			// at this point we are not currently "parsing" a known type from the string, therfore the next character should 
			// decide what type is next. 
		
			IF Path[currentCharacterPositionInPath] = DOLLAR_SIGN THEN
				
				// i.e. the following string $.myValue would indicate that we are here.
				//                           ^                                         
				// as such, we do not need to take any action.  We already create a root element at the start, so this is an 
				// optional character which they do not need to supply. 				
				
			ELSIF Path[currentCharacterPositionInPath] = PERIOD THEN
				
				// i.e. the following string $.myValue would indicate that we are here.
				//                            ^                                        
				// as such, we do not need to take any action.  
				
			ELSIF Path[currentCharacterPositionInPath] = LEFT_SQUARE_BRACKET THEN
				
				// i.e. the following string $.myValue[1].['myProperty'] would indicate that we could be at the start of one of two types
				//                                    ^   ^                                      
				// as such, we mark that we could be either a property or array and continue				
				currentlyParsingType := BRACKET_NOTATION_PROPERTY_OR_ARRAY;				
				
			ELSIF Path[currentCharacterPositionInPath] = RIGHT_SQUARE_BRACKET THEN
				
				// This would indicate a failed parse as this should not happen.
				JsonPathVisitor.InvalidSyntaxFound(RIGHT_SQUARE_BRACKET, currentCharacterPositionInPath);
				
			ELSIF Path[currentCharacterPositionInPath] = SINGLE_QUOTE THEN
				
				// This would indicate a failed parse as this should not happen.
				JsonPathVisitor.InvalidSyntaxFound(SINGLE_QUOTE, currentCharacterPositionInPath);
				
			ELSE
				
				// i.e. the following string $.myValue[1].['myProperty'] would indicate that we could be at the start of a property
				//                             ^                      
				currentlyParsingType := DOT_NOTATION_PROPERTY;
				currentElementStart := currentCharacterPositionInPath;	
		
			END_IF
			
		DOT_NOTATION_PROPERTY:
		
			IF Path[currentCharacterPositionInPath] = PERIOD OR Path[currentCharacterPositionInPath] = LEFT_SQUARE_BRACKET OR Path[currentCharacterPositionInPath] = NULL THEN
				
				currentElementEnd := currentCharacterPositionInPath - 1;
				
				currentElementLength := 1 + currentElementEnd - currentElementStart;
				memset(ADR(elementText),0,SIZEOF(elementText));
				memcpy(ADR(elementText),ADR(Path[currentElementStart]),currentElementLength);
		
				JsonPathVisitor.PropertyFound(elementText);
				
				currentlyParsingType := NOTHING;
				CONTINUE;
				
			END_IF
			
		BRACKET_NOTATION_PROPERTY_OR_ARRAY:
		
			IF Path[currentCharacterPositionInPath] = SINGLE_QUOTE THEN
				currentlyParsingType := BRACKET_NOTATION_PROPERTY_ELEMENT;
				currentElementStart := currentCharacterPositionInPath + 1;			
			ELSE
				currentlyParsingType := BRACKET_NOTATION_ARRAY_ELEMENT;
				currentElementStart := currentCharacterPositionInPath;			
			END_IF
			
		BRACKET_NOTATION_PROPERTY_ELEMENT:
		
			IF Path[currentCharacterPositionInPath] = SINGLE_QUOTE THEN
				
				currentElementEnd := currentCharacterPositionInPath - 1;

				currentElementLength := 1 + currentElementEnd - currentElementStart;
				memset(ADR(elementText),0,SIZEOF(elementText));
				memcpy(ADR(elementText),ADR(Path[currentElementStart]),currentElementLength);
				
				JsonPathVisitor.PropertyFound(elementText);
			
				currentlyParsingType := NOTHING;
						
			END_IF
			
		BRACKET_NOTATION_ARRAY_ELEMENT:
		
			IF Path[currentCharacterPositionInPath] = RIGHT_SQUARE_BRACKET THEN
				
				currentElementEnd := currentCharacterPositionInPath - 1;
				
				currentElementLength := 1 + currentElementEnd - currentElementStart;
				memset(ADR(elementText),0,SIZEOF(elementText));
				memcpy(ADR(elementText),ADR(Path[currentElementStart]),currentElementLength);
				
				JsonPathVisitor.ArrayIndexFound(STRING_TO_UDINT(elementText));		
				currentlyParsingType := NOTHING;
						
			END_IF
			

	END_CASE
	
	currentCharacterPositionInPath := currentCharacterPositionInPath + 1;
	
UNTIL endOfRepeat 
END_REPEAT

JsonPathVisitor.EndOfParse();
END_METHOD

END_FUNCTION_BLOCK

// mobject-json/_Internal/JsonPathVisitor/I_JsonPathVisitor
INTERFACE I_JsonPathVisitor EXTENDS __System.IQueryInterface

METHOD ArrayIndexFound
VAR_INPUT
	Index : UDINT;
END_VAR
END_METHOD

METHOD EndOfParse
VAR_INPUT
END_VAR
END_METHOD

METHOD InvalidSyntaxFound
VAR_INPUT
	Character : BYTE;
	Position : UDINT;
END_VAR
END_METHOD

METHOD PropertyFound
VAR_INPUT
	Name : T_MAXSTRING;
END_VAR
END_METHOD

METHOD StartOfParse
VAR_INPUT
END_VAR
END_METHOD

END_INTERFACE

// mobject-json/_Internal/JsonPathVisitor/JsonDomNavigator
{attribute 'linkalways'} 
{attribute 'no_explicit_call' := 'This FB is a CLASS and must be accessed using methods or properties'}
{attribute 'enable_dynamic_creation'}
FUNCTION_BLOCK JsonDomNavigator IMPLEMENTS I_JsonPathVisitor
VAR
	jsonDomParser : REFERENCE TO JsonDomParser;
	currentJsonPosition : SJsonValue;
	_currentNode : SJsonValue;
END_VAR

METHOD FB_init : BOOL
VAR_INPUT
	bInitRetains : BOOL; // if TRUE, the retain variables are initialized (warm start / cold start)
	bInCopyCode : BOOL;  // if TRUE, the instance afterwards gets moved into the copy code (online change)
	JsonDomParser : REFERENCE TO JsonDomParser;
END_VAR
THIS^.jsonDomParser REF= JsonDomParser;
END_METHOD

METHOD ArrayIndexFound
VAR_INPUT
	Index : UDINT;
END_VAR
currentJsonPosition := jsonDomParser.GetArrayValueByIdx(currentJsonPosition, Index);
END_METHOD

PROPERTY PUBLIC CurrentNode : SJsonValue
GET
CurrentNode := _currentNode;
END_GET
END_PROPERTY

METHOD EndOfParse
VAR_INPUT
END_VAR
_currentNode := currentJsonPosition;
END_METHOD

METHOD InvalidSyntaxFound
VAR_INPUT
	Character : BYTE;
	Position : UDINT;
END_VAR
currentJsonPosition := 0;
END_METHOD

METHOD PropertyFound
VAR_INPUT
	Name : T_MAXSTRING;
END_VAR
currentJsonPosition := jsonDomParser.FindMember(currentJsonPosition,Name);
END_METHOD

METHOD StartOfParse
VAR_INPUT
END_VAR
currentJsonPosition := jsonDomParser.GetDocumentRoot();
END_METHOD

END_FUNCTION_BLOCK

// mobject-json/_Internal/JsonPathVisitor/JsonDomCreator
{attribute 'linkalways'} 
{attribute 'no_explicit_call' := 'This FB is a CLASS and must be accessed using methods or properties'}
{attribute 'enable_dynamic_creation'}
FUNCTION_BLOCK JsonDomCreator IMPLEMENTS I_JsonPathVisitor
VAR
	jsonDomParser : REFERENCE TO JsonDomParser;
	currentJsonPosition : SJsonValue;
	_currentNode : SJsonValue;
END_VAR

METHOD FB_init : BOOL
VAR_INPUT
	bInitRetains : BOOL; // if TRUE, the retain variables are initialized (warm start / cold start)
	bInCopyCode : BOOL;  // if TRUE, the instance afterwards gets moved into the copy code (online change)
	JsonDomParser : REFERENCE TO JsonDomParser;
END_VAR
THIS^.jsonDomParser REF= JsonDomParser;
END_METHOD

METHOD PRIVATE PadStartOfArray : SJsonValue
VAR_INPUT
	Index : UDINT;
	ArrayPosition : SJsonValue;
END_VAR
VAR
	i : UDINT;
	arrayValueLocation : SJsonValue;
END_VAR
FOR i := 0 TO Index DO
		
	arrayValueLocation := jsonDomParser.GetArrayValueByIdx(ArrayPosition, Index);
	IF arrayValueLocation <> 0 THEN
		CONTINUE;
	END_IF
	
	arrayValueLocation := jsonDomParser.PushbackNullValue(ArrayPosition);

END_FOR

PadStartOfArray := arrayValueLocation;
END_METHOD

METHOD ArrayIndexFound
VAR_INPUT
	Index : UDINT;
END_VAR
VAR
	memberLocation : SJsonValue;
	i : UDINT;
END_VAR
IF jsonDomParser.IsArray(currentJsonPosition) THEN
	
	memberLocation := jsonDomParser.GetArrayValueByIdx(currentJsonPosition, Index);
	
	IF memberLocation <> 0 THEN
		currentJsonPosition := memberLocation;
		RETURN;
	END_IF
	
	currentJsonPosition := PadStartOfArray(Index, currentJsonPosition);

else
	
	memberLocation := jsonDomParser.SetArray(currentJsonPosition,0);
	currentJsonPosition := PadStartOfArray(Index, memberLocation);
	
END_IF
END_METHOD

PROPERTY PUBLIC CurrentNode : SJsonValue
GET
CurrentNode := _currentNode;
END_GET
END_PROPERTY

METHOD EndOfParse
VAR_INPUT
END_VAR
_currentNode := currentJsonPosition;
END_METHOD

METHOD InvalidSyntaxFound
VAR_INPUT
	Character : BYTE;
	Position : UDINT;
END_VAR
currentJsonPosition := 0;
END_METHOD

METHOD PropertyFound
VAR_INPUT
	Name : T_MAXSTRING;
END_VAR
VAR
	memberLocation : SJsonValue;
END_VAR
memberLocation := jsonDomParser.FindMember(currentJsonPosition,Name);

IF memberLocation <> 0 THEN
	currentJsonPosition := memberLocation;
	RETURN;
END_IF

currentJsonPosition := jsonDomParser.AddNullMember(currentJsonPosition,Name);
END_METHOD

METHOD StartOfParse
VAR_INPUT
END_VAR
currentJsonPosition := jsonDomParser.GetDocumentRoot();
END_METHOD

END_FUNCTION_BLOCK

// mobject-json/_Internal/JsonDeserializerNode/JsonDeserializerNode
{attribute 'linkalways'} 
{attribute 'no_explicit_call' := 'This FB is a CLASS and must be accessed using methods or properties'}
{attribute 'enable_dynamic_creation'}
FUNCTION_BLOCK JsonDeserializerNode EXTENDS Disposable IMPLEMENTS I_Deserializer
VAR	
	parent : I_JsonDeserializer;
	jsonParser : REFERENCE TO JsonDomParser;
	root : SJsonValue;
	garbageCollector : I_DeserializerGarbageCollector;
	nullNode : I_Deserializer;
	errorFactory : DeserializationErrorFactory;
END_VAR

METHOD FB_init : BOOL
VAR_INPUT
	bInitRetains : BOOL; // if TRUE, the retain variables are initialized (warm start / cold start)
	bInCopyCode : BOOL;  // if TRUE, the instance afterwards gets moved into the copy code (online change)
	ParentJsonDeserializer : I_JsonDeserializer;
	ParentJsonDomParser : REFERENCE TO JsonDomParser;
	NodeRoot : SJsonValue;
	ParentGarbageCollector : I_DeserializerGarbageCollector;
	ParentNullDeserializer : I_Deserializer;
END_VAR
THIS^.parent := ParentJsonDeserializer;
THIS^.jsonParser REF= ParentJsonDomParser;
THIS^.root := NodeRoot;
THIS^.garbageCollector := ParentGarbageCollector;
THIS^.nullNode := ParentNullDeserializer;

ParentGarbageCollector.Register(THIS^);
END_METHOD

METHOD PROTECTED CreateArrayForwardEnumerator : I_DeserializerArrayForwardEnumerator
VAR_INPUT
	DeserializerRoot : SJsonValue;
END_VAR
VAR 
	pForwardEnumerator : POINTER TO JsonDeserializerArrayForwardEnumerator;
END_VAR
pForwardEnumerator := __NEW(JsonDeserializerArrayForwardEnumerator(
	ParentJsonDeserializer := parent,
	ParentJsonDomParser := jsonParser, 
	NodeRoot := DeserializerRoot, 
	ParentGarbageCollector := garbageCollector, 
	ParentNullDeserializer := nullNode
));

CreateArrayForwardEnumerator := pForwardEnumerator^;
END_METHOD

METHOD PROTECTED CreateDeserializer : I_Deserializer
VAR_INPUT
	DeserializerRoot : SJsonValue;
END_VAR
VAR 
	pNode : POINTER TO JsonDeserializerNode;
END_VAR
pNode := __NEW(JsonDeserializerNode(
	ParentJsonDeserializer := parent,
	ParentJsonDomParser := jsonParser, 
	NodeRoot := DeserializerRoot, 
	ParentGarbageCollector := garbageCollector, 
	ParentNullDeserializer := nullNode
));

CreateDeserializer := pNode^;
END_METHOD

METHOD PROTECTED CreateObjectForwardEnumerator : I_DeserializerObjectForwardEnumerator
VAR_INPUT
	DeserializerRoot : SJsonValue;
END_VAR
VAR 
	pForwardEnumerator : POINTER TO JsonDeserializerObjectForwardEnumerator;
END_VAR
pForwardEnumerator := __NEW(JsonDeserializerObjectForwardEnumerator(
	ParentJsonDeserializer := parent,
	ParentJsonDomParser := jsonParser, 
	NodeRoot := DeserializerRoot, 
	ParentGarbageCollector := garbageCollector, 
	ParentNullDeserializer := nullNode
));

CreateObjectForwardEnumerator := pForwardEnumerator^;
END_METHOD

METHOD PROTECTED TryGetMember : BOOL
VAR_INPUT
	MemberName : T_MAXSTRING;
	Member : REFERENCE TO SJsonValue;
	Feedback : I_DeserializerFeedback;
END_VAR
VAR
	localMember : SJsonValue;
	error : I_Error;
END_VAR
IF MemberName = '' THEN
	error := errorFactory.CreateInvalidKeyError();
	Feedback.LogError(error);
	RETURN;
END_IF

localMember := jsonParser.FindMember(root, MemberName);

IF localMember = 0 THEN
	error := errorFactory.CreateMissingKeyError(MemberName);
	Feedback.LogError(error);
	RETURN;
END_IF

Member := localMember;
TryGetMember := TRUE;
END_METHOD

METHOD PROTECTED TryReadBool : BOOL
VAR_INPUT
	JsonValue : SJsonValue;
	Destination : ANY;
END_VAR
VAR
	_BOOL : BOOL;
END_VAR
IF jsonValue = 0 THEN
	RETURN;
END_IF

IF jsonParser.IsBool(jsonValue) THEN
	_BOOL := jsonParser.GetBool(jsonValue);
	TryReadBool := TryConvert_BOOL_TO_DESTINATION(_BOOL,Destination);
	RETURN;
END_IF
END_METHOD

METHOD PROTECTED TryReadNumber : BOOL
VAR_INPUT
	JsonValue : SJsonValue;
	Destination : ANY;
END_VAR
VAR
	_DINT : DINT;
	_LINT : LINT;
	_UDINT : UDINT;
	_ULINT : ULINT;
	_LREAL : LREAL;
END_VAR
IF jsonValue = 0 THEN
	RETURN;
END_IF

IF jsonParser.IsInt(jsonValue) THEN
	_DINT := jsonParser.GetInt(jsonValue);
	TryReadNumber := TryConvert_DINT_TO_DESTINATION(_DINT,Destination);
	RETURN;
END_IF

IF jsonParser.IsInt64(jsonValue) THEN
	_LINT := jsonParser.GetInt64(jsonValue);
	TryReadNumber := TryConvert_LINT_TO_DESTINATION(_LINT,Destination);
	RETURN;
END_IF

IF jsonParser.IsUInt(jsonValue) THEN
	_UDINT := jsonParser.GetUInt(jsonValue);
	TryReadNumber := TryConvert_UDINT_TO_DESTINATION(_UDINT,Destination);
	RETURN;
END_IF

IF jsonParser.IsUInt64(jsonValue) THEN
	_ULINT := jsonParser.GetUInt64(jsonValue);
	TryReadNumber := TryConvert_ULINT_TO_DESTINATION(_ULINT,Destination);
	RETURN;
END_IF

IF jsonParser.IsDouble(jsonValue) THEN
	_LREAL := jsonParser.GetDouble(jsonValue);
	TryReadNumber := TryConvert_LREAL_TO_DESTINATION(_LREAL,Destination);
	RETURN;
END_IF
END_METHOD

METHOD PROTECTED TryReadString : BOOL
VAR_INPUT
	JsonValue : SJsonValue;
	Destination : REFERENCE TO STRING;
END_VAR
IF jsonValue = 0 THEN
	RETURN;
END_IF

IF jsonParser.IsString(jsonValue) THEN
	IF (jsonParser.CopyString(jsonValue,Destination,DINT_TO_UDINT(SIZEOF(Destination))) > 0) THEN;
		TryReadString := TRUE;
		RETURN;
	END_IF
END_IF
END_METHOD

METHOD PUBLIC Clone : I_Deserializer
VAR
	pClone : POINTER TO JsonDeserializer;
	jsonSize : UDINT;
	pJsonString : POINTER TO STRING;
END_VAR
pClone := __NEW(JsonDeserializer);
Clone := pClone^;

jsonSize := jsonParser.GetJsonLength(root);

IF jsonSize = 0 THEN
	// no further cloning to do. 
	RETURN;
END_IF

pJsonString := __NEW(BYTE, jsonSize);

IF jsonParser.CopyJson(root, pJsonString^, jsonSize) = 0 THEN
	__DELETE(pJsonString);
	RETURN;
END_IF

pClone^.TryLoad(pJsonString^);
__DELETE(pJsonString);
END_METHOD

METHOD Dispose
VAR
END_VAR
garbageCollector.Deregister(THIS^);
super^.Dispose();
END_METHOD

METHOD GetArray : I_Deserializer
IF NOT jsonParser.IsArray(root) THEN
	GetArray := nullNode;
	RETURN;
END_IF

GetArray := CreateDeserializer(root);
END_METHOD

METHOD GetArrayEnumerator : I_DeserializerArrayForwardEnumerator
VAR_INPUT
END_VAR
GetArrayEnumerator := CreateArrayForwardEnumerator(root);
END_METHOD

METHOD GetElementByIndex : I_Deserializer
VAR_INPUT
	Index : UDINT;
END_VAR
VAR
	newRoot : SJsonValue;
END_VAR
IF NOT jsonParser.IsArray(root) THEN
	GetElementByIndex := nullNode;
	RETURN;
END_IF

newRoot := jsonParser.GetArrayValueByIdx(root, Index);

IF newRoot = 0 THEN
	GetElementByIndex := nullNode;
	RETURN;
END_IF

GetElementByIndex := CreateDeserializer(newRoot);
END_METHOD

METHOD GetKeyArray : I_Deserializer
VAR_INPUT
	Key : T_MAXSTRING;
END_VAR
VAR
	member : SJsonValue;
END_VAR
IF key = '' THEN
	RETURN;
END_IF

member := jsonParser.FindMember(root,Key);

IF member = 0 THEN
	GetKeyArray := nullNode;
	RETURN;
END_IF

IF NOT jsonParser.IsArray(member) THEN
	GetKeyArray := nullNode;
	RETURN;
END_IF

GetKeyArray := CreateDeserializer(member);
END_METHOD

METHOD GetKeyObject : I_Deserializer
VAR_INPUT
	Key : T_MAXSTRING;
END_VAR
VAR
	newRoot : SJsonValue;
END_VAR
newRoot := jsonParser.FindMember(root, Key);

IF newRoot = 0 THEN
	GetKeyObject := nullNode;
	RETURN;
END_IF

GetKeyObject := CreateDeserializer(newRoot);
END_METHOD

METHOD GetObject : I_Deserializer
IF NOT jsonParser.IsObject(root) THEN
	GetObject := nullNode;
	RETURN;
END_IF

GetObject := CreateDeserializer(root);
END_METHOD

METHOD GetObjectEnumerator : I_DeserializerObjectForwardEnumerator
VAR_INPUT
END_VAR
GetObjectEnumerator := CreateObjectForwardEnumerator(root);
END_METHOD

METHOD GetValue : I_Deserializer
VAR
	newRoot : SJsonValue;
END_VAR
newRoot := jsonParser.GetMemberValue(root);

IF newRoot = 0 THEN
	GetValue := nullNode;
	RETURN;
END_IF

GetValue := CreateDeserializer(newRoot);
END_METHOD

METHOD TryDeserializeKeyToObject : BOOL
VAR_INPUT
	Key : T_MAXSTRING;
	Object : I_Deserializable;
	Feedback : I_DeserializerFeedback;
END_VAR
VAR
	member : SJsonValue;
	error : I_Error;
	deserializer : I_Deserializer;
END_VAR
IF NOT TryGetMember(Key, member, Feedback) THEN
	RETURN;
END_IF

deserializer := CreateDeserializer(member);
TryDeserializeKeyToObject := Object.TryDeserializeFrom(deserializer, Feedback);
END_METHOD

METHOD TryDeserializeToObject : BOOL
VAR_INPUT
	Object : I_Deserializable;
	Feedback : I_DeserializerFeedback;
END_VAR
TryDeserializeToObject := Object.TryDeserializeFrom(THIS^, Feedback);
END_METHOD

METHOD TryGetBase64 : BOOL
VAR_INPUT
	pBytes : POINTER TO BYTE;
	nBytes : DINT;
	Feedback : I_DeserializerFeedback;
END_VAR
VAR
	error : I_Error;
END_VAR
IF NOT jsonParser.IsBase64(root) THEN
	error := errorFactory.CreateIncorrectTypeError('Base64');
	Feedback.LogError(error);
	RETURN;
END_IF

jsonParser.GetBase64(root, pBytes, nBytes);
TryGetBase64 := TRUE;
END_METHOD

METHOD TryGetBool : BOOL
VAR_INPUT
	Destination : REFERENCE TO BOOL;
	Feedback : I_DeserializerFeedback;
END_VAR
VAR
	value : BOOL;
	error : I_Error;
END_VAR
IF NOT TryReadBool(root, value) THEN
	error := errorFactory.CreateIncorrectTypeError('BOOL');
	Feedback.LogError(error);
	RETURN;
END_IF

Destination := value;
TryGetBool := TRUE;
END_METHOD

METHOD TryGetByte : BOOL
VAR_INPUT
	Destination : REFERENCE TO BYTE;
	Feedback : I_DeserializerFeedback;
END_VAR
VAR
	value : BYTE;
	error : I_Error;
END_VAR
IF NOT TryReadNumber(root, value) THEN
	error := errorFactory.CreateIncorrectTypeError('BYTE');
	Feedback.LogError(error);
	RETURN;
END_IF

Destination := value;
TryGetByte := TRUE;
END_METHOD

METHOD TryGetDateTime : BOOL
VAR_INPUT
	Destination : REFERENCE TO DATE_AND_TIME;
	Feedback : I_DeserializerFeedback;
END_VAR
VAR
	error : I_Error;
END_VAR
IF NOT jsonParser.IsISO8601TimeFormat(root) THEN
	error := errorFactory.CreateIncorrectTypeError('DATE_AND_TIME');
	Feedback.LogError(error);
	RETURN;
END_IF

Destination := jsonParser.GetDateTime(root);
TryGetDateTime := TRUE;
END_METHOD

METHOD TryGetDcTime : BOOL
VAR_INPUT
	Destination : REFERENCE TO DCTIME;
	Feedback : I_DeserializerFeedback;
END_VAR
VAR
	error : I_Error;
END_VAR
IF NOT jsonParser.IsISO8601TimeFormat(root) THEN
	error := errorFactory.CreateIncorrectTypeError('DCTIME');
	Feedback.LogError(error);
	RETURN;
END_IF

Destination := jsonParser.GetDcTime(root);
TryGetDcTime := TRUE;
END_METHOD

METHOD TryGetDint : BOOL
VAR_INPUT
	Destination : REFERENCE TO DINT;
	Feedback : I_DeserializerFeedback;
END_VAR
VAR
	value : DINT;
	error : I_Error;
END_VAR
IF NOT TryReadNumber(root, value) THEN
	error := errorFactory.CreateIncorrectTypeError('DINT');
	Feedback.LogError(error);
	RETURN;
END_IF

Destination := value;
TryGetDint := TRUE;
END_METHOD

METHOD TryGetDword : BOOL
VAR_INPUT
	Destination : REFERENCE TO DWORD;
	Feedback : I_DeserializerFeedback;
END_VAR
VAR
	value : DWORD;
	error : I_Error;
END_VAR
IF NOT TryReadNumber(root, value) THEN
	error := errorFactory.CreateIncorrectTypeError('DWORD');
	Feedback.LogError(error);
	RETURN;
END_IF

Destination := value;
TryGetDword := TRUE;
END_METHOD

METHOD TryGetFileTime : BOOL
VAR_INPUT
	Destination : REFERENCE TO FILETIME;
	Feedback : I_DeserializerFeedback;
END_VAR
VAR
	error : I_Error;
END_VAR
IF NOT jsonParser.IsISO8601TimeFormat(root) THEN
	error := errorFactory.CreateIncorrectTypeError('FILETIME');
	Feedback.LogError(error);
	RETURN;
END_IF

Destination := jsonParser.GetFileTime(root);
TryGetFileTime := TRUE;
END_METHOD

METHOD TryGetHexAsBytes : BOOL
VAR_INPUT
	pBytes : POINTER TO BYTE;
	nBytes : DINT;
	Feedback : I_DeserializerFeedback;
END_VAR
VAR
	error : I_Error;
END_VAR
IF NOT jsonParser.IsHexBinary(root) THEN
	error := errorFactory.CreateIncorrectTypeError('HexBinary');
	Feedback.LogError(error);
	RETURN;
END_IF

jsonParser.GetHexBinary(root, pBytes, nBytes);
TryGetHexAsBytes := TRUE;
END_METHOD

METHOD TryGetInt : BOOL
VAR_INPUT
	Destination : REFERENCE TO INT;
	Feedback : I_DeserializerFeedback;
END_VAR
VAR
	value : INT;
	error : I_Error;
END_VAR
IF NOT TryReadNumber(root, value) THEN
	error := errorFactory.CreateIncorrectTypeError('INT');
	Feedback.LogError(error);
	RETURN;
END_IF

Destination := value;
TryGetInt := TRUE;
END_METHOD

METHOD TryGetKeyBase64 : BOOL
VAR_INPUT
	Key : T_MAXSTRING;
	pBytes : POINTER TO BYTE;
	nBytes : DINT;
	Feedback : I_DeserializerFeedback;
END_VAR
VAR
	member : SJsonValue;
	error : I_Error;
END_VAR
IF NOT TryGetMember(Key, member, Feedback) THEN
	RETURN;
END_IF

IF NOT jsonParser.IsBase64(member) THEN
	error := errorFactory.CreateIncorrectKeyTypeError('Base64',Key);
	Feedback.LogError(error);
	RETURN;
END_IF

jsonParser.GetBase64(member, pBytes, nBytes);
TryGetKeyBase64 := TRUE;
END_METHOD

METHOD TryGetKeyBool : BOOL
VAR_INPUT
	Key : T_MAXSTRING;
	Destination : REFERENCE TO BOOL;
	Feedback : I_DeserializerFeedback;
END_VAR
VAR
	member : SJsonValue;
	value : BOOL;
	error : I_Error;
END_VAR
IF NOT TryGetMember(Key, member, Feedback) THEN
	RETURN;
END_IF

IF NOT TryReadBool(member, value) THEN
	error := errorFactory.CreateIncorrectKeyTypeError('BOOL',Key);
	Feedback.LogError(error);
	RETURN;
END_IF

Destination := value;
TryGetKeyBool := TRUE;
END_METHOD

METHOD TryGetKeyByte : BOOL
VAR_INPUT
	Key : T_MAXSTRING;
	Destination : REFERENCE TO BYTE;
	Feedback : I_DeserializerFeedback;
END_VAR
VAR
	value : BYTE;
	member : SJsonValue;
	error : I_Error;
END_VAR
IF NOT TryGetMember(Key, member, Feedback) THEN
	RETURN;
END_IF

IF NOT TryReadNumber(member, value) THEN
	error := errorFactory.CreateIncorrectKeyTypeError('BYTE',Key);
	Feedback.LogError(error);
	RETURN;
END_IF

Destination := value;
TryGetKeyByte := TRUE;
END_METHOD

METHOD TryGetKeyDateTime : BOOL
VAR_INPUT
	Key : T_MAXSTRING;
	Destination : REFERENCE TO DATE_AND_TIME;
	Feedback : I_DeserializerFeedback;
END_VAR
VAR
	member : SJSonValue;
	error : I_Error;
END_VAR
IF NOT TryGetMember(Key, member, Feedback) THEN
	RETURN;
END_IF

IF NOT jsonParser.IsISO8601TimeFormat(member) THEN
	error := errorFactory.CreateIncorrectKeyTypeError('DATE_AND_TIME',Key);
	Feedback.LogError(error);
	RETURN;
END_IF

Destination := jsonParser.GetDateTime(member);
TryGetKeyDateTime := TRUE;
END_METHOD

METHOD TryGetKeyDcTime : BOOL
VAR_INPUT
	Key : T_MAXSTRING;
	Destination : REFERENCE TO DCTIME;
	Feedback : I_DeserializerFeedback;
END_VAR
VAR
	member : SJSonValue;
	error : I_Error;
END_VAR
IF NOT TryGetMember(Key, member, Feedback) THEN
	RETURN;
END_IF

IF NOT jsonParser.IsISO8601TimeFormat(member) THEN
	error := errorFactory.CreateIncorrectKeyTypeError('DCTIME',Key);
	Feedback.LogError(error);
	RETURN;
END_IF

Destination := jsonParser.GetDcTime(member);
TryGetKeyDcTime := TRUE;
END_METHOD

METHOD TryGetKeyDint : BOOL
VAR_INPUT
	Key : T_MAXSTRING;
	Destination : REFERENCE TO DINT;
	Feedback : I_DeserializerFeedback;
END_VAR
VAR
	member : SJsonValue;
	value : DINT;
	error : I_Error;
END_VAR
IF NOT TryGetMember(Key, member, Feedback) THEN
	RETURN;
END_IF

IF NOT TryReadNumber(member, value) THEN
	error := errorFactory.CreateIncorrectKeyTypeError('DINT',Key);
	Feedback.LogError(error);
	RETURN;
END_IF

Destination := value;
TryGetKeyDint := TRUE;
END_METHOD

METHOD TryGetKeyDword : BOOL
VAR_INPUT
	Key : T_MAXSTRING;
	Destination : REFERENCE TO DWORD;
	Feedback : I_DeserializerFeedback;
END_VAR
VAR
	member : SJsonValue;
	value : DWORD;
	error : I_Error;
END_VAR
IF NOT TryGetMember(Key, member, Feedback) THEN
	RETURN;
END_IF

IF NOT TryReadNumber(member, value) THEN
	error := errorFactory.CreateIncorrectKeyTypeError('DWORD',Key);
	Feedback.LogError(error);
	RETURN;
END_IF

Destination := value;
TryGetKeyDword := TRUE;
END_METHOD

METHOD TryGetKeyFileTime : BOOL
VAR_INPUT
	Key : T_MAXSTRING;
	Destination : REFERENCE TO FILETIME;
	Feedback : I_DeserializerFeedback;
END_VAR
VAR
	member : SJSonValue;
	error : I_Error;
END_VAR
IF NOT TryGetMember(Key, member, Feedback) THEN
	RETURN;
END_IF

IF NOT jsonParser.IsISO8601TimeFormat(member) THEN
	error := errorFactory.CreateIncorrectKeyTypeError('FILETIME',Key);
	Feedback.LogError(error);
	RETURN;
END_IF

Destination := jsonParser.GetFileTime(member);
TryGetKeyFileTime := TRUE;
END_METHOD

METHOD TryGetKeyHexAsBytes : BOOL
VAR_INPUT
	Key : T_MAXSTRING;
	pBytes : POINTER TO BYTE;
	nBytes : DINT;
	Feedback : I_DeserializerFeedback;
END_VAR
VAR
	member : SJsonValue;
	error : I_Error;
END_VAR
IF NOT TryGetMember(Key, member, Feedback) THEN
	RETURN;
END_IF

IF NOT jsonParser.IsHexBinary(member) THEN
	error := errorFactory.CreateIncorrectKeyTypeError('HexBinary',Key);
	Feedback.LogError(error);
	RETURN;
END_IF

jsonParser.GetHexBinary(member, pBytes, nBytes);
TryGetKeyHexAsBytes := TRUE;
END_METHOD

METHOD TryGetKeyInt : BOOL
VAR_INPUT
	Key : T_MAXSTRING;
	Destination : REFERENCE TO INT;
	Feedback : I_DeserializerFeedback;
END_VAR
VAR
	member : SJsonValue;
	value : INT;
	error : I_Error;
END_VAR
IF NOT TryGetMember(Key, member, Feedback) THEN
	RETURN;
END_IF

IF NOT TryReadNumber(member, value) THEN
	error := errorFactory.CreateIncorrectKeyTypeError('INT',Key);
	Feedback.LogError(error);
	RETURN;
END_IF

Destination := value;
TryGetKeyInt := TRUE;
END_METHOD

METHOD TryGetKeyLint : BOOL
VAR_INPUT
	Key : T_MAXSTRING;
	Destination : REFERENCE TO LINT;
	Feedback : I_DeserializerFeedback;
END_VAR
VAR
	member : SJsonValue;
	value : LINT;
	error : I_Error;
END_VAR
IF NOT TryGetMember(Key, member, Feedback) THEN
	RETURN;
END_IF

IF NOT TryReadNumber(member, value) THEN
	error := errorFactory.CreateIncorrectKeyTypeError('LINT',Key);
	Feedback.LogError(error);
	RETURN;
END_IF

Destination := value;
TryGetKeyLint := TRUE;
END_METHOD

METHOD TryGetKeyLreal : BOOL
VAR_INPUT
	Key : T_MAXSTRING;
	Destination : REFERENCE TO LREAL;
	Feedback : I_DeserializerFeedback;
END_VAR
VAR
	member : SJsonValue;
	value : LREAL;
	error : I_Error;
END_VAR
IF NOT TryGetMember(Key, member, Feedback) THEN
	RETURN;
END_IF

IF NOT TryReadNumber(member, value) THEN
	error := errorFactory.CreateIncorrectKeyTypeError('LREAL',Key);
	Feedback.LogError(error);
	RETURN;
END_IF

Destination := value;
TryGetKeyLreal := TRUE;
END_METHOD

METHOD TryGetKeyLtime : BOOL
VAR_INPUT
	Key : T_MAXSTRING;
	Destination : REFERENCE TO LTIME;
	Feedback : I_DeserializerFeedback;
END_VAR
VAR
	member : SJsonValue;
	timeAsString : T_MAXSTRING;
	error : I_Error;
END_VAR
IF NOT TryGetMember(Key, member, Feedback) THEN
	RETURN;
END_IF

IF NOT jsonParser.IsString(member) THEN
	error := errorFactory.CreateIncorrectKeyTypeError('LTIME',Key);
	Feedback.LogError(error);
	RETURN;
END_IF

timeAsString := jsonParser.GetString(member);
Destination := STRING_TO_LTIME(timeAsString);

TryGetKeyLtime := TRUE;
END_METHOD

METHOD TryGetKeyLword : BOOL
VAR_INPUT
	Key : T_MAXSTRING;
	Destination : REFERENCE TO LWORD;
	Feedback : I_DeserializerFeedback;
END_VAR
VAR
	member : SJsonValue;
	value : LWORD;
	error : I_Error;
END_VAR
IF NOT TryGetMember(Key, member, Feedback) THEN
	RETURN;
END_IF

IF NOT TryReadNumber(member, value) THEN
	error := errorFactory.CreateIncorrectKeyTypeError('LWORD',Key);
	Feedback.LogError(error);
	RETURN;
END_IF

Destination := value;
TryGetKeyLword := TRUE;
END_METHOD

METHOD TryGetKeyReal : BOOL
VAR_INPUT
	Key : T_MAXSTRING;
	Destination : REFERENCE TO REAL;
	Feedback : I_DeserializerFeedback;
END_VAR
VAR
	member : SJsonValue;
	value : REAL;
	error : I_Error;
END_VAR
IF NOT TryGetMember(Key, member, Feedback) THEN
	RETURN;
END_IF

IF NOT TryReadNumber(member, value) THEN
	error := errorFactory.CreateIncorrectKeyTypeError('REAL',Key);
	Feedback.LogError(error);
	RETURN;
END_IF

Destination := value;
TryGetKeyReal := TRUE;
END_METHOD

METHOD TryGetKeySint : BOOL
VAR_INPUT
	Key : T_MAXSTRING;
	Destination : REFERENCE TO SINT;
	Feedback : I_DeserializerFeedback;
END_VAR
VAR
	member : SJsonValue;
	value : SINT;
	error : I_Error;
END_VAR
IF NOT TryGetMember(Key, member, Feedback) THEN
	RETURN;
END_IF

IF NOT TryReadNumber(member, value) THEN
	error := errorFactory.CreateIncorrectKeyTypeError('SINT',Key);
	Feedback.LogError(error);
	RETURN;
END_IF

Destination := value;
TryGetKeySint := TRUE;
END_METHOD

METHOD TryGetKeyString : BOOL
VAR_INPUT
	Key : T_MAXSTRING;
	Destination : REFERENCE TO STRING;
	Feedback : I_DeserializerFeedback;
END_VAR
VAR
	member : SJsonValue;
	error : I_Error;
END_VAR
IF NOT TryGetMember(Key, member, Feedback) THEN
	RETURN;
END_IF

IF NOT TryReadString(member, Destination) THEN
	error := errorFactory.CreateIncorrectKeyTypeError('STRING',Key);
	Feedback.LogError(error);
	RETURN;
END_IF

TryGetKeyString := TRUE;
END_METHOD

METHOD TryGetKeyTime : BOOL
VAR_INPUT
	Key : T_MAXSTRING;
	Destination : REFERENCE TO TIME;
	Feedback : I_DeserializerFeedback;
END_VAR
VAR
	member : SJsonValue;
	timeAsString : T_MAXSTRING;
	error : I_Error;
END_VAR
IF NOT TryGetMember(Key, member, Feedback) THEN
	RETURN;
END_IF

IF NOT jsonParser.IsString(member) THEN
	error := errorFactory.CreateIncorrectKeyTypeError('TIME',Key);
	Feedback.LogError(error);
	RETURN;
END_IF

timeAsString := jsonParser.GetString(member);
Destination := STRING_TO_TIME(timeAsString);

TryGetKeyTime := TRUE;
END_METHOD

METHOD TryGetKeyTod : BOOL
VAR_INPUT
	Key : T_MAXSTRING;
	Destination : REFERENCE TO TOD;
	Feedback : I_DeserializerFeedback;
END_VAR
VAR
	member : SJsonValue;
	timeAsString : T_MAXSTRING;
	error : I_Error;
END_VAR
IF NOT TryGetMember(Key, member, Feedback) THEN
	RETURN;
END_IF

IF NOT jsonParser.IsString(member) THEN
	error := errorFactory.CreateIncorrectKeyTypeError('TOD',Key);
	Feedback.LogError(error);
	RETURN;
END_IF

timeAsString := jsonParser.GetString(member);
Destination := STRING_TO_TOD(timeAsString);

TryGetKeyTod := TRUE;
END_METHOD

METHOD TryGetKeyUdint : BOOL
VAR_INPUT
	Key : T_MAXSTRING;
	Destination : REFERENCE TO UDINT;
	Feedback : I_DeserializerFeedback;
END_VAR
VAR
	member : SJsonValue;
	value : UDINT;
	error : I_Error;
END_VAR
IF NOT TryGetMember(Key, member, Feedback) THEN
	RETURN;
END_IF

IF NOT TryReadNumber(member, value) THEN
	error := errorFactory.CreateIncorrectKeyTypeError('UDINT',Key);
	Feedback.LogError(error);
	RETURN;
END_IF

Destination := value;
TryGetKeyUdint := TRUE;
END_METHOD

METHOD TryGetKeyUint : BOOL
VAR_INPUT
	Key : T_MAXSTRING;
	Destination : REFERENCE TO UINT;
	Feedback : I_DeserializerFeedback;
END_VAR
VAR
	member : SJsonValue;
	value : UINT;
	error : I_Error;
END_VAR
IF NOT TryGetMember(Key, member, Feedback) THEN
	RETURN;
END_IF

IF NOT TryReadNumber(member, value) THEN
	error := errorFactory.CreateIncorrectKeyTypeError('UINT',Key);
	Feedback.LogError(error);
	RETURN;
END_IF

Destination := value;
TryGetKeyUint := TRUE;
END_METHOD

METHOD TryGetKeyUlint : BOOL
VAR_INPUT
	Key : T_MAXSTRING;
	Destination : REFERENCE TO ULINT;
	Feedback : I_DeserializerFeedback;
END_VAR
VAR
	member : SJsonValue;
	value : ULINT;
	error : I_Error;
END_VAR
IF NOT TryGetMember(Key, member, Feedback) THEN
	RETURN;
END_IF

IF NOT TryReadNumber(member, value) THEN
	error := errorFactory.CreateIncorrectKeyTypeError('ULINT',Key);
	Feedback.LogError(error);
	RETURN;
END_IF

Destination := value;
TryGetKeyUlint := TRUE;
END_METHOD

METHOD TryGetKeyUsint : BOOL
VAR_INPUT
	Key : T_MAXSTRING;
	Destination : REFERENCE TO USINT;
	Feedback : I_DeserializerFeedback;
END_VAR
VAR
	member : SJsonValue;
	value : USINT;
	error : I_Error;
END_VAR
IF NOT TryGetMember(Key, member, Feedback) THEN
	RETURN;
END_IF

IF NOT TryReadNumber(member, value) THEN
	error := errorFactory.CreateIncorrectKeyTypeError('USINT',Key);
	Feedback.LogError(error);
	RETURN;
END_IF

Destination := value;
TryGetKeyUsint := TRUE;
END_METHOD

METHOD TryGetKeyWord : BOOL
VAR_INPUT
	Key : T_MAXSTRING;
	Destination : REFERENCE TO WORD;
	Feedback : I_DeserializerFeedback;
END_VAR
VAR
	member : SJsonValue;
	value : WORD;
	error : I_Error;
END_VAR
IF NOT TryGetMember(Key, member, Feedback) THEN
	RETURN;
END_IF

IF NOT TryReadNumber(member, value) THEN
	error := errorFactory.CreateIncorrectKeyTypeError('USINT',Key);
	Feedback.LogError(error);
	RETURN;
END_IF

Destination := value;
TryGetKeyWord := TRUE;
END_METHOD

METHOD TryGetLint : BOOL
VAR_INPUT
	Destination : REFERENCE TO LINT;
	Feedback : I_DeserializerFeedback;
END_VAR
VAR
	value : LINT;
	error : I_Error;
END_VAR
IF NOT TryReadNumber(root, value) THEN
	error := errorFactory.CreateIncorrectTypeError('LINT');
	Feedback.LogError(error);
	RETURN;
END_IF

Destination := value;
TryGetLint := TRUE;
END_METHOD

METHOD TryGetLreal : BOOL
VAR_INPUT
	Destination : REFERENCE TO LREAL;
	Feedback : I_DeserializerFeedback;
END_VAR
VAR
	value : LREAL;
	error : I_Error;
END_VAR
IF NOT TryReadNumber(root, value) THEN
	error := errorFactory.CreateIncorrectTypeError('LREAL');
	Feedback.LogError(error);
	RETURN;
END_IF

Destination := value;
TryGetLreal := TRUE;
END_METHOD

METHOD TryGetLtime : BOOL
VAR_INPUT
	Destination : REFERENCE TO LTIME;
	Feedback : I_DeserializerFeedback;
END_VAR
VAR
	timeAsString : T_MAXSTRING;
	error : I_Error;
END_VAR
IF NOT jsonParser.IsString(root) THEN
	error := errorFactory.CreateIncorrectTypeError('LTIME');
	Feedback.LogError(error);
	RETURN;
END_IF

timeAsString := jsonParser.GetString(root);
Destination := STRING_TO_LTIME(timeAsString);

TryGetLtime := TRUE;
END_METHOD

METHOD TryGetLword : BOOL
VAR_INPUT
	Destination : REFERENCE TO LWORD;
	Feedback : I_DeserializerFeedback;
END_VAR
VAR
	value : LWORD;
	error : I_Error;
END_VAR
IF NOT TryReadNumber(root, value) THEN
	error := errorFactory.CreateIncorrectTypeError('LWORD');
	Feedback.LogError(error);
	RETURN;
END_IF

Destination := value;
TryGetLword := TRUE;
END_METHOD

METHOD TryGetReal : BOOL
VAR_INPUT
	Destination : REFERENCE TO REAL;
	Feedback : I_DeserializerFeedback;
END_VAR
VAR
	value : REAL;
	error : I_Error;
END_VAR
IF NOT TryReadNumber(root, value) THEN
	error := errorFactory.CreateIncorrectTypeError('REAL');
	Feedback.LogError(error);
	RETURN;
END_IF

Destination := value;
TryGetReal := TRUE;
END_METHOD

METHOD TryGetSint : BOOL
VAR_INPUT
	Destination : REFERENCE TO SINT;
	Feedback : I_DeserializerFeedback;
END_VAR
VAR
	value : SINT;
	error : I_Error;
END_VAR
IF NOT TryReadNumber(root, value) THEN
	error := errorFactory.CreateIncorrectTypeError('SINT');
	Feedback.LogError(error);
	RETURN;
END_IF

Destination := value;
TryGetSint := TRUE;
END_METHOD

METHOD TryGetString : BOOL
VAR_INPUT
	Destination : REFERENCE TO STRING;
	Feedback : I_DeserializerFeedback;
END_VAR
VAR
	error : I_Error;
END_VAR
IF NOT jsonParser.IsString(root) THEN
	error := errorFactory.CreateIncorrectTypeError('STRING');
	Feedback.LogError(error);
	RETURN;
END_IF

Destination := jsonParser.GetString(root);
TryGetString := TRUE;
END_METHOD

METHOD TryGetTime : BOOL
VAR_INPUT
	Destination : REFERENCE TO TIME;
	Feedback : I_DeserializerFeedback;
END_VAR
VAR
	timeAsString : T_MAXSTRING;
	error : I_Error;
END_VAR
IF NOT jsonParser.IsString(root) THEN
	error := errorFactory.CreateIncorrectTypeError('TIME');
	Feedback.LogError(error);
	RETURN;
END_IF

timeAsString := jsonParser.GetString(root);
Destination := STRING_TO_TIME(timeAsString);

TryGetTime := TRUE;
END_METHOD

METHOD TryGetTod : BOOL
VAR_INPUT
	Destination : REFERENCE TO TOD;
	Feedback : I_DeserializerFeedback;
END_VAR
VAR
	timeAsString : T_MAXSTRING;
	error : I_Error;
END_VAR
IF NOT jsonParser.IsString(root) THEN
	error := errorFactory.CreateIncorrectTypeError('TOD');
	Feedback.LogError(error);
	RETURN;
END_IF

timeAsString := jsonParser.GetString(root);
Destination := STRING_TO_TOD(timeAsString);

TryGetTod := TRUE;
END_METHOD

METHOD TryGetUdint : BOOL
VAR_INPUT
	Destination : REFERENCE TO UDINT;
	Feedback : I_DeserializerFeedback;
END_VAR
VAR
	value : UDINT;
	error : I_Error;
END_VAR
IF NOT TryReadNumber(root, value) THEN
	error := errorFactory.CreateIncorrectTypeError('UDINT');
	Feedback.LogError(error);
	RETURN;
END_IF

Destination := value;
TryGetUdint := TRUE;
END_METHOD

METHOD TryGetUint : BOOL
VAR_INPUT
	Destination : REFERENCE TO UINT;
	Feedback : I_DeserializerFeedback;
END_VAR
VAR
	value : UINT;
	error : I_Error;
END_VAR
IF NOT TryReadNumber(root, value) THEN
	error := errorFactory.CreateIncorrectTypeError('UINT');
	Feedback.LogError(error);
	RETURN;
END_IF

Destination := value;
TryGetUint := TRUE;
END_METHOD

METHOD TryGetUlint : BOOL
VAR_INPUT
	Destination : REFERENCE TO ULINT;
	Feedback : I_DeserializerFeedback;
END_VAR
VAR
	value : ULINT;
	error : I_Error;
END_VAR
IF NOT TryReadNumber(root, value) THEN
	error := errorFactory.CreateIncorrectTypeError('ULINT');
	Feedback.LogError(error);
	RETURN;
END_IF

Destination := value;
TryGetUlint := TRUE;
END_METHOD

METHOD TryGetUsint : BOOL
VAR_INPUT
	Destination : REFERENCE TO USINT;
	Feedback : I_DeserializerFeedback;
END_VAR
VAR
	value : USINT;
	error : I_Error;
END_VAR
IF NOT TryReadNumber(root, value) THEN
	error := errorFactory.CreateIncorrectTypeError('USINT');
	Feedback.LogError(error);
	RETURN;
END_IF

Destination := value;
TryGetUsint := TRUE;
END_METHOD

METHOD TryGetWord : BOOL
VAR_INPUT
	Destination : REFERENCE TO WORD;
	Feedback : I_DeserializerFeedback;
END_VAR
VAR
	value : WORD;
	error : I_Error;
END_VAR
IF NOT TryReadNumber(root, value) THEN
	error := errorFactory.CreateIncorrectTypeError('WORD');
	Feedback.LogError(error);
	RETURN;
END_IF

Destination := value;
TryGetWord := TRUE;
END_METHOD

END_FUNCTION_BLOCK

// mobject-json/_Internal/JsonDeserializerForwardEnumerator/JsonDeserializerObjectForwardEnumerator
{attribute 'linkalways'} 
{attribute 'no_explicit_call' := 'This FB is a CLASS and must be accessed using methods or properties'}
{attribute 'enable_dynamic_creation'}
FUNCTION_BLOCK JsonDeserializerObjectForwardEnumerator EXTENDS Disposable IMPLEMENTS I_DeserializerObjectForwardEnumerator, I_EventHandler
VAR
	parent : I_JsonDeserializer;
	jsonParser : REFERENCE TO JsonDomParser;
	root : SJsonValue;
	garbageCollector : I_DeserializerGarbageCollector;
	nullNode : I_Deserializer;
	moveNextCalled : BOOL := FALSE;
	invalid : BOOL := FALSE; 
	nextMemberPosition : SJsonValue;
	memberBeginPosition : SJsonValue;
	memberEndPosition : SJsonValue;
	currentDeserializer : I_Deserializer;
	currentKey : T_MAXSTRING;
END_VAR

METHOD FB_init : BOOL
VAR_INPUT
	bInitRetains : BOOL; // if TRUE, the retain variables are initialized (warm start / cold start)
	bInCopyCode : BOOL;  // if TRUE, the instance afterwards gets moved into the copy code (online change)
	ParentJsonDeserializer : I_JsonDeserializer;
	ParentJsonDomParser : REFERENCE TO JsonDomParser;
	NodeRoot : SJsonValue;
	ParentGarbageCollector : I_DeserializerGarbageCollector;
	ParentNullDeserializer : I_Deserializer;
END_VAR
THIS^.parent := ParentJsonDeserializer;
THIS^.jsonParser REF= ParentJsonDomParser;
THIS^.root := NodeRoot;
THIS^.garbageCollector := ParentGarbageCollector;
THIS^.nullNode := ParentNullDeserializer;

Initialize();

Parent.OnEvent('OnChanged',THIS^);
Parent.OnEvent('OnDisposed',THIS^);
END_METHOD

METHOD FB_exit : BOOL
VAR_INPUT
	bInCopyCode : BOOL; // if TRUE, the exit method is called for exiting an instance that is copied afterwards (online change).
END_VAR
IF bInCopyCode THEN
	RETURN;
END_IF

IF parent = 0 THEN
	RETURN;
END_IF

parent.OffEvent('OnChanged',THIS^);
parent.OffEvent('OnDisposed',THIS^);
END_METHOD

METHOD PROTECTED CreateDeserializer : I_Deserializer
VAR_INPUT
	DeserializerRoot : SJsonValue;
END_VAR
VAR 
	pNode : POINTER TO JsonDeserializerNode;
END_VAR
pNode := __NEW(JsonDeserializerNode(
	ParentJsonDeserializer := parent,
	ParentJsonDomParser := jsonParser, 
	NodeRoot := DeserializerRoot, 
	ParentGarbageCollector := garbageCollector, 
	ParentNullDeserializer := nullNode
));

CreateDeserializer := pNode^;
END_METHOD

METHOD PROTECTED Initialize
VAR_INPUT
END_VAR
IF NOT jsonParser.IsObject(root) THEN
	invalid := TRUE;
	RETURN;
END_IF

memberBeginPosition := jsonParser.MemberBegin(root);
memberEndPosition := jsonParser.MemberEnd(root);

IF memberBeginPosition = 0 THEN
	invalid := TRUE;
	RETURN;
END_IF

IF memberEndPosition = 0 THEN
	invalid := TRUE;
	RETURN;
END_IF
END_METHOD

METHOD PROTECTED UpdateCurrentDeserializer
VAR_INPUT
	UpdatedRoot : SJsonValue;
END_VAR
VAR
	rootOfValue : SJsonValue;
END_VAR
IF currentDeserializer <> 0 THEN
	currentDeserializer.Dispose();
	currentDeserializer := 0;
END_IF

IF invalid THEN
	RETURN;
END_IF

rootOfValue := jsonParser.GetMemberValue(UpdatedRoot);
currentKey := jsonParser.GetMemberName(UpdatedRoot);

IF rootOfValue = 0 THEN
	RETURN;
END_IF

currentDeserializer := CreateDeserializer(rootOfValue);
END_METHOD

PROPERTY PUBLIC Current : I_Deserializer
GET
IF NOT IsValid THEN
	Current := nullNode;
	RETURN;
END_IF

IF currentDeserializer = 0 THEN
	Current := nullNode;
	RETURN;
END_IF

Current := currentDeserializer;
END_GET
END_PROPERTY

METHOD PUBLIC HandleEvent
VAR_INPUT
	Event : I_Event;
END_VAR
VAR
	changedEvent : I_JsonDeserializerChangedEvent;
	disposedEvent : I_JsonDeserializerDisposedEvent;
END_VAR
IF __QUERYINTERFACE(Event, changedEvent) THEN
	invalid := TRUE;
ELSIF __QUERYINTERFACE(Event, disposedEvent) THEN
	parent := 0;
	Dispose();
END_IF
END_METHOD

PROPERTY PUBLIC IsValid : BOOL
GET
PUBLIC
IF invalid THEN
	RETURN;
END_IF

IF parent = 0 THEN
	RETURN;
END_IF

IsValid := TRUE;
END_GET
END_PROPERTY

PROPERTY Key : T_MAXSTRING
GET
Key := currentKey;
END_GET
END_PROPERTY

METHOD PUBLIC MoveNext : BOOL
IF invalid THEN
    RETURN;
END_IF

// Handle the initial move
IF NOT moveNextCalled THEN
    moveNextCalled := TRUE;
    UpdateCurrentDeserializer(memberBeginPosition);
	nextMemberPosition := jsonParser.NextMember(memberBeginPosition);
	MoveNext := TRUE;
    RETURN;
END_IF

// Handle subsequent moves
IF nextMemberPosition <> memberEndPosition THEN	
	UpdateCurrentDeserializer(nextMemberPosition);
	nextMemberPosition := jsonParser.NextMember(nextMemberPosition);
	MoveNext := TRUE;
END_IF
END_METHOD

END_FUNCTION_BLOCK

// mobject-json/JsonDeserializer/JsonDeserializer
{attribute 'linkalways'} 
{attribute 'no_explicit_call' := 'This FB is a CLASS and must be accessed using methods or properties'}
{attribute 'enable_dynamic_creation'}
FUNCTION_BLOCK JsonDeserializer EXTENDS Disposable IMPLEMENTS I_JsonDeserializer
VAR
	jsonParser : JsonDomParser;
	root : SJsonValue;
	garbageCollector : DeserializerGarbageCollector;
	nullNode : JsonDeserializerNullNode(THIS^);
	rootNode : I_Deserializer := nullNode;
	eventEmitter : EventEmitter;
END_VAR

METHOD FB_exit : BOOL
VAR_INPUT
	bInCopyCode : BOOL; // if TRUE, the exit method is called for exiting an instance that is copied afterwards (online change).
END_VAR
IF bInCopyCode THEN
	RETURN;
END_IF

Reset();
EmitDisposedEvent();
END_METHOD

METHOD PROTECTED CreateDeserializer : I_Deserializer
VAR_INPUT
	DeserializerRoot : SJsonValue;
END_VAR
VAR 
	pNode : POINTER TO JsonDeserializerNode;
END_VAR
pNode := __NEW(JsonDeserializerNode(
	ParentJsonDeserializer := THIS^,
	ParentJsonDomParser := jsonParser, 
	NodeRoot := DeserializerRoot, 
	ParentGarbageCollector := garbageCollector, 
	ParentNullDeserializer := nullNode)
);

CreateDeserializer := pNode^;
END_METHOD

METHOD PRIVATE EmitChangedEvent
VAR
	pJsonDeserializerChangedEvent : POINTER TO JsonDeserializerChangedEvent;
END_VAR
pJsonDeserializerChangedEvent := __NEW(JsonDeserializerChangedEvent(Target := THIS^));
eventEmitter.Emit('OnChanged', pJsonDeserializerChangedEvent^);
pJsonDeserializerChangedEvent^.Dispose();
END_METHOD

METHOD PRIVATE EmitDisposedEvent
VAR
	pJsonDeserializerDisposedEvent : POINTER TO JsonDeserializerDisposedEvent;
END_VAR
pJsonDeserializerDisposedEvent := __NEW(JsonDeserializerDisposedEvent(Target := THIS^));
eventEmitter.Emit('OnDisposed', pJsonDeserializerDisposedEvent^);
pJsonDeserializerDisposedEvent^.Dispose();
END_METHOD

METHOD PUBLIC Clone : I_Deserializer
VAR
	pClone : POINTER TO JsonDeserializer;
	jsonSize : UDINT;
	pJsonString : POINTER TO STRING;
END_VAR
pClone := __NEW(JsonDeserializer);
Clone := pClone^;

jsonSize := jsonParser.GetDocumentLength();

IF jsonSize = 0 THEN
	// no further cloning to do. 
	RETURN;
END_IF

pJsonString := __NEW(BYTE, jsonSize);

IF jsonParser.CopyDocument(pJsonString^, jsonSize) = 0 THEN
	__DELETE(pJsonString);
	RETURN;
END_IF

pClone^.TryLoad(pJsonString^);
__DELETE(pJsonString);
END_METHOD

METHOD GetArray : I_Deserializer
VAR_INPUT
END_VAR
GetArray := rootNode.GetArray();
END_METHOD

METHOD GetArrayEnumerator : I_DeserializerArrayForwardEnumerator
VAR_INPUT
END_VAR
GetArrayEnumerator := rootNode.GetArrayEnumerator();
END_METHOD

METHOD GetElementByIndex : I_Deserializer
VAR_INPUT
	Index : UDINT;
END_VAR
GetElementByIndex := rootNode.GetElementByIndex(Index);
END_METHOD

METHOD GetKeyArray : I_Deserializer
VAR_INPUT
	Key : T_MAXSTRING;
END_VAR
GetKeyArray := rootNode.GetKeyArray(Key);
END_METHOD

METHOD GetKeyObject : I_Deserializer
VAR_INPUT
	Key : T_MAXSTRING;
END_VAR
GetKeyObject := rootNode.GetKeyObject(Key);
END_METHOD

METHOD GetObject : I_Deserializer
VAR_INPUT
END_VAR
GetObject := rootNode.GetObject();
END_METHOD

METHOD GetObjectEnumerator : I_DeserializerObjectForwardEnumerator
VAR_INPUT
END_VAR
GetObjectEnumerator := rootNode.GetObjectEnumerator();
END_METHOD

METHOD PUBLIC OffEvent
VAR_INPUT
	EventName : T_MaxString;
	EventHandler : I_EventHandler;
END_VAR
eventEmitter.OffEvent(EventName, EventHandler);
END_METHOD

METHOD PUBLIC OnceEvent
VAR_INPUT
	EventName : T_MaxString;
	EventHandler : I_EventHandler;
END_VAR
eventEmitter.OnceEvent(EventName, EventHandler);
END_METHOD

METHOD PUBLIC OnEvent
VAR_INPUT
	EventName : T_MaxString;
	EventHandler : I_EventHandler;
END_VAR
eventEmitter.OnEvent(EventName, EventHandler);
END_METHOD

METHOD PUBLIC Reset
VAR_INPUT
END_VAR
jsonParser.NewDocument();
garbageCollector.Execute();
root := 0;
rootNode := nullNode;
EmitChangedEvent();
END_METHOD

METHOD TryDeserializeKeyToObject : BOOL
VAR_INPUT
	Key : T_MAXSTRING;
	Object : I_Deserializable;
	Feedback : I_DeserializerFeedback;
END_VAR
TryDeserializeKeyToObject := rootNode.TryDeserializeKeyToObject(Key,Object, Feedback);
END_METHOD

METHOD TryDeserializeToObject : BOOL
VAR_INPUT
	Object : I_Deserializable;
	Feedback : I_DeserializerFeedback;
END_VAR
TryDeserializeToObject := rootNode.TryDeserializeToObject(Object, Feedback);
END_METHOD

METHOD TryGetBase64 : BOOL
VAR_INPUT
	pBytes : POINTER TO BYTE;
	nBytes : DINT;
	Feedback : I_DeserializerFeedback;
END_VAR
TryGetBase64 := rootNode.TryGetBase64(pBytes, nBytes, Feedback);
END_METHOD

METHOD TryGetBool : BOOL
VAR_INPUT
	Destination : REFERENCE TO BOOL;
	Feedback : I_DeserializerFeedback;
END_VAR
TryGetBool := rootNode.TryGetBool(Destination, Feedback);
END_METHOD

METHOD TryGetByte : BOOL
VAR_INPUT
	Destination : REFERENCE TO BYTE;
	Feedback : I_DeserializerFeedback;
END_VAR
TryGetByte := rootNode.TryGetByte(Destination, Feedback);
END_METHOD

METHOD TryGetDateTime : BOOL
VAR_INPUT
	Destination : REFERENCE TO DATE_AND_TIME;
	Feedback : I_DeserializerFeedback;
END_VAR
TryGetDateTime := rootNode.TryGetDateTime(Destination, Feedback);
END_METHOD

METHOD TryGetDcTime : BOOL
VAR_INPUT
	Destination : REFERENCE TO DCTIME;
	Feedback : I_DeserializerFeedback;
END_VAR
TryGetDcTime := rootNode.TryGetDcTime(Destination, Feedback);
END_METHOD

METHOD TryGetDint : BOOL
VAR_INPUT
	Destination : REFERENCE TO DINT;
	Feedback : I_DeserializerFeedback;
END_VAR
TryGetDint := rootNode.TryGetDint(Destination, Feedback);
END_METHOD

METHOD TryGetDword : BOOL
VAR_INPUT
	Destination : REFERENCE TO DWORD;
	Feedback : I_DeserializerFeedback;
END_VAR
TryGetDword := rootNode.TryGetDword(Destination, Feedback);
END_METHOD

METHOD TryGetFileTime : BOOL
VAR_INPUT
	Destination : REFERENCE TO FILETIME;
	Feedback : I_DeserializerFeedback;
END_VAR
TryGetFileTime := rootNode.TryGetFileTime(Destination, Feedback);
END_METHOD

METHOD TryGetHexAsBytes : BOOL
VAR_INPUT
	pBytes : POINTER TO BYTE;
	nBytes : DINT;
	Feedback : I_DeserializerFeedback;
END_VAR
TryGetHexAsBytes := rootNode.TryGetHexAsBytes(pBytes, nBytes, Feedback);
END_METHOD

METHOD TryGetInt : BOOL
VAR_INPUT
	Destination : REFERENCE TO INT;
	Feedback : I_DeserializerFeedback;
END_VAR
TryGetInt := rootNode.TryGetInt(Destination, Feedback);
END_METHOD

METHOD TryGetKeyBase64 : BOOL
VAR_INPUT
	Key : T_MAXSTRING;
	pBytes : POINTER TO BYTE;
	nBytes : DINT;
	Feedback : I_DeserializerFeedback;
END_VAR
TryGetKeyBase64 := rootNode.TryGetKeyBase64(Key, pBytes, nBytes, Feedback);
END_METHOD

METHOD TryGetKeyBool : BOOL
VAR_INPUT
	Key : T_MAXSTRING;
	Destination : REFERENCE TO BOOL;
	Feedback : I_DeserializerFeedback;
END_VAR
TryGetKeyBool := rootNode.TryGetKeyBool(Key, Destination, Feedback);
END_METHOD

METHOD TryGetKeyByte : BOOL
VAR_INPUT
	Key : T_MAXSTRING;
	Destination : REFERENCE TO BYTE;
	Feedback : I_DeserializerFeedback;
END_VAR
TryGetKeyByte := rootNode.TryGetKeyByte(Key, Destination, Feedback);
END_METHOD

METHOD TryGetKeyDateTime : BOOL
VAR_INPUT
	Key : T_MAXSTRING;
	Destination : REFERENCE TO DATE_AND_TIME;
	Feedback : I_DeserializerFeedback;
END_VAR
TryGetKeyDateTime := rootNode.TryGetKeyDateTime(Key, Destination, Feedback);
END_METHOD

METHOD TryGetKeyDcTime : BOOL
VAR_INPUT
	Key : T_MAXSTRING;
	Destination : REFERENCE TO DCTIME;
	Feedback : I_DeserializerFeedback;
END_VAR
TryGetKeyDcTime := rootNode.TryGetKeyDcTime(Key, Destination, Feedback);
END_METHOD

METHOD TryGetKeyDint : BOOL
VAR_INPUT
	Key : T_MAXSTRING;
	Destination : REFERENCE TO DINT;
	Feedback : I_DeserializerFeedback;
END_VAR
TryGetKeyDint := rootNode.TryGetKeyDint(Key, Destination, Feedback);
END_METHOD

METHOD TryGetKeyDword : BOOL
VAR_INPUT
	Key : T_MAXSTRING;
	Destination : REFERENCE TO DWORD;
	Feedback : I_DeserializerFeedback;
END_VAR
TryGetKeyDword := rootNode.TryGetKeyDword(Key, Destination, Feedback);
END_METHOD

METHOD TryGetKeyFileTime : BOOL
VAR_INPUT
	Key : T_MAXSTRING;
	Destination : REFERENCE TO FILETIME;
	Feedback : I_DeserializerFeedback;
END_VAR
TryGetKeyFileTime := rootNode.TryGetKeyFileTime(Key, Destination, Feedback);
END_METHOD

METHOD TryGetKeyHexAsBytes : BOOL
VAR_INPUT
	Key : T_MAXSTRING;
	pBytes : POINTER TO BYTE;
	nBytes : DINT;
	Feedback : I_DeserializerFeedback;
END_VAR
TryGetKeyHexAsBytes := rootNode.TryGetKeyHexAsBytes(Key, pBytes, nBytes, Feedback);
END_METHOD

METHOD TryGetKeyInt : BOOL
VAR_INPUT
	Key : T_MAXSTRING;
	Destination : REFERENCE TO INT;
	Feedback : I_DeserializerFeedback;
END_VAR
TryGetKeyInt := rootNode.TryGetKeyInt(Key, Destination, Feedback);
END_METHOD

METHOD TryGetKeyLint : BOOL
VAR_INPUT
	Key : T_MAXSTRING;
	Destination : REFERENCE TO LINT;
	Feedback : I_DeserializerFeedback;
END_VAR
TryGetKeyLint := rootNode.TryGetKeyLint(Key, Destination, Feedback);
END_METHOD

METHOD TryGetKeyLreal : BOOL
VAR_INPUT
	Key : T_MAXSTRING;
	Destination : REFERENCE TO LREAL;
	Feedback : I_DeserializerFeedback;
END_VAR
TryGetKeyLreal := rootNode.TryGetKeyLreal(Key, Destination, Feedback);
END_METHOD

METHOD TryGetKeyLtime : BOOL
VAR_INPUT
	Key : T_MAXSTRING;
	Destination : REFERENCE TO LTIME;
	Feedback : I_DeserializerFeedback;
END_VAR
TryGetKeyLtime := rootNode.TryGetKeyLtime(Key, Destination, Feedback);
END_METHOD

METHOD TryGetKeyLword : BOOL
VAR_INPUT
	Key : T_MAXSTRING;
	Destination : REFERENCE TO LWORD;
	Feedback : I_DeserializerFeedback;
END_VAR
TryGetKeyLword := rootNode.TryGetKeyLword(Key, Destination, Feedback);
END_METHOD

METHOD TryGetKeyReal : BOOL
VAR_INPUT
	Key : T_MAXSTRING;
	Destination : REFERENCE TO REAL;
	Feedback : I_DeserializerFeedback;
END_VAR
TryGetKeyReal := rootNode.TryGetKeyReal(Key, Destination, Feedback);
END_METHOD

METHOD TryGetKeySint : BOOL
VAR_INPUT
	Key : T_MAXSTRING;
	Destination : REFERENCE TO SINT;
	Feedback : I_DeserializerFeedback;
END_VAR
TryGetKeySint := rootNode.TryGetKeySint(Key, Destination, Feedback);
END_METHOD

METHOD TryGetKeyString : BOOL
VAR_INPUT
	Key : T_MAXSTRING;
	Destination : REFERENCE TO STRING;
	Feedback : I_DeserializerFeedback;
END_VAR
TryGetKeyString := rootNode.TryGetKeyString(Key, Destination, Feedback);
END_METHOD

METHOD TryGetKeyTime : BOOL
VAR_INPUT
	Key : T_MAXSTRING;
	Destination : REFERENCE TO TIME;
	Feedback : I_DeserializerFeedback;
END_VAR
TryGetKeyTime := rootNode.TryGetKeyTime(Key, Destination, Feedback);
END_METHOD

METHOD TryGetKeyTod : BOOL
VAR_INPUT
	Key : T_MAXSTRING;
	Destination : REFERENCE TO TOD;
	Feedback : I_DeserializerFeedback;
END_VAR
TryGetKeyTod := rootNode.TryGetKeyTod(Key, Destination, Feedback);
END_METHOD

METHOD TryGetKeyUdint : BOOL
VAR_INPUT
	Key : T_MAXSTRING;
	Destination : REFERENCE TO UDINT;
	Feedback : I_DeserializerFeedback;
END_VAR
TryGetKeyUdint := rootNode.TryGetKeyUdint(Key, Destination, Feedback);
END_METHOD

METHOD TryGetKeyUint : BOOL
VAR_INPUT
	Key : T_MAXSTRING;
	Destination : REFERENCE TO UINT;
	Feedback : I_DeserializerFeedback;
END_VAR
TryGetKeyUint := rootNode.TryGetKeyUint(Key, Destination, Feedback);
END_METHOD

METHOD TryGetKeyUlint : BOOL
VAR_INPUT
	Key : T_MAXSTRING;
	Destination : REFERENCE TO ULINT;
	Feedback : I_DeserializerFeedback;
END_VAR
TryGetKeyUlint := rootNode.TryGetKeyUlint(Key, Destination, Feedback);
END_METHOD

METHOD TryGetKeyUsint : BOOL
VAR_INPUT
	Key : T_MAXSTRING;
	Destination : REFERENCE TO USINT;
	Feedback : I_DeserializerFeedback;
END_VAR
TryGetKeyUsint := rootNode.TryGetKeyUsint(Key, Destination, Feedback);
END_METHOD

METHOD TryGetKeyWord : BOOL
VAR_INPUT
	Key : T_MAXSTRING;
	Destination : REFERENCE TO WORD;
	Feedback : I_DeserializerFeedback;
END_VAR
TryGetKeyWord := rootNode.TryGetKeyWord(Key, Destination, Feedback);
END_METHOD

METHOD TryGetLint : BOOL
VAR_INPUT
	Destination : REFERENCE TO LINT;
	Feedback : I_DeserializerFeedback;
END_VAR
TryGetLint := rootNode.TryGetLint(Destination, Feedback);
END_METHOD

METHOD TryGetLreal : BOOL
VAR_INPUT
	Destination : REFERENCE TO LREAL;
	Feedback : I_DeserializerFeedback;
END_VAR
TryGetLreal := rootNode.TryGetLreal(Destination, Feedback);
END_METHOD

METHOD TryGetLtime : BOOL
VAR_INPUT
	Destination : REFERENCE TO LTIME;
	Feedback : I_DeserializerFeedback;
END_VAR
TryGetLtime := rootNode.TryGetLtime(Destination, Feedback);
END_METHOD

METHOD TryGetLword : BOOL
VAR_INPUT
	Destination : REFERENCE TO LWORD;
	Feedback : I_DeserializerFeedback;
END_VAR
TryGetLword := rootNode.TryGetLword(Destination, Feedback);
END_METHOD

METHOD TryGetReal : BOOL
VAR_INPUT
	Destination : REFERENCE TO REAL;
	Feedback : I_DeserializerFeedback;
END_VAR
TryGetReal := rootNode.TryGetReal(Destination, Feedback);
END_METHOD

METHOD TryGetSint : BOOL
VAR_INPUT
	Destination : REFERENCE TO SINT;
	Feedback : I_DeserializerFeedback;
END_VAR
TryGetSint := rootNode.TryGetSint(Destination, Feedback);
END_METHOD

METHOD TryGetString : BOOL
VAR_INPUT
	Destination : REFERENCE TO STRING;
	Feedback : I_DeserializerFeedback;
END_VAR
TryGetString := rootNode.TryGetString(Destination, Feedback);
END_METHOD

METHOD TryGetTime : BOOL
VAR_INPUT
	Destination : REFERENCE TO TIME;
	Feedback : I_DeserializerFeedback;
END_VAR
TryGetTime := rootNode.TryGetTime(Destination, Feedback);
END_METHOD

METHOD TryGetTod : BOOL
VAR_INPUT
	Destination : REFERENCE TO TOD;
	Feedback : I_DeserializerFeedback;
END_VAR
TryGetTod := rootNode.TryGetTod(Destination, Feedback);
END_METHOD

METHOD TryGetUdint : BOOL
VAR_INPUT
	Destination : REFERENCE TO UDINT;
	Feedback : I_DeserializerFeedback;
END_VAR
TryGetUdint := rootNode.TryGetUdint(Destination, Feedback);
END_METHOD

METHOD TryGetUint : BOOL
VAR_INPUT
	Destination : REFERENCE TO UINT;
	Feedback : I_DeserializerFeedback;
END_VAR
TryGetUint := rootNode.TryGetUint(Destination, Feedback);
END_METHOD

METHOD TryGetUlint : BOOL
VAR_INPUT
	Destination : REFERENCE TO ULINT;
	Feedback : I_DeserializerFeedback;
END_VAR
TryGetUlint := rootNode.TryGetUlint(Destination, Feedback);
END_METHOD

METHOD TryGetUsint : BOOL
VAR_INPUT
	Destination : REFERENCE TO USINT;
	Feedback : I_DeserializerFeedback;
END_VAR
TryGetUsint := rootNode.TryGetUsint(Destination, Feedback);
END_METHOD

METHOD TryGetWord : BOOL
VAR_INPUT
	Destination : REFERENCE TO WORD;
	Feedback : I_DeserializerFeedback;
END_VAR
TryGetWord := rootNode.TryGetWord(Destination, Feedback);
END_METHOD

METHOD PUBLIC TryLoad : BOOL
VAR_INPUT
	SerializedData : REFERENCE TO STRING;;
END_VAR
Reset();
EmitChangedEvent();

root := jsonParser.ParseDocument(SerializedData);
IF root = 0 THEN
	RETURN;
END_IF

rootNode := CreateDeserializer(root);
TryLoad := TRUE;
END_METHOD

END_FUNCTION_BLOCK

// mobject-json/_Internal/JsonDeserializerNode/JsonDeserializerNullNode
{attribute 'linkalways'} 
{attribute 'no_explicit_call' := 'This FB is a CLASS and must be accessed using methods or properties'}
{attribute 'enable_dynamic_creation'}
FUNCTION_BLOCK JsonDeserializerNullNode EXTENDS Disposable IMPLEMENTS I_Deserializer
VAR
	parent : I_JsonDeserializer;
	errorFactory : DeserializationErrorFactory;
END_VAR

METHOD FB_init : BOOL
VAR_INPUT
	bInitRetains : BOOL; // if TRUE, the retain variables are initialized (warm start / cold start)
	bInCopyCode : BOOL;  // if TRUE, the instance afterwards gets moved into the copy code (online change)
	ParentJsonDeserializer : I_JsonDeserializer;
END_VAR
THIS^.parent := ParentJsonDeserializer;
END_METHOD

METHOD PROTECTED CreateNullArrayEnumerator : I_DeserializerArrayForwardEnumerator
VAR_INPUT
END_VAR
VAR
	pForwardEnumerator : POINTER TO JsonDeserializerNullArrayForwardEnumerator;
END_VAR
pForwardEnumerator := __NEW(JsonDeserializerNullArrayForwardEnumerator(ParentJsonDeserializer := parent, ParentNullDeserializer := THIS^));
CreateNullArrayEnumerator := pForwardEnumerator^;
END_METHOD

METHOD PROTECTED CreateNullObjectEnumerator : I_DeserializerObjectForwardEnumerator
VAR_INPUT
END_VAR
VAR
	pForwardEnumerator : POINTER TO JsonDeserializerNullObjectForwardEnumerator;
END_VAR
pForwardEnumerator := __NEW(JsonDeserializerNullObjectForwardEnumerator(ParentJsonDeserializer := parent, ParentNullDeserializer := THIS^));
CreateNullObjectEnumerator := pForwardEnumerator^;
END_METHOD

METHOD PUBLIC Clone : I_Deserializer
VAR
	pClone : POINTER TO JsonDeserializerNullNode;
END_VAR
pClone := __NEW(JsonDeserializerNullNode(ParentJsonDeserializer := parent));
Clone := pClone^;
END_METHOD

METHOD GetArray : I_Deserializer
VAR_INPUT
END_VAR
GetArray := this^;
END_METHOD

METHOD GetArrayEnumerator : I_DeserializerArrayForwardEnumerator
VAR_INPUT
END_VAR
GetArrayEnumerator := CreateNullArrayEnumerator();
END_METHOD

METHOD GetElementByIndex : I_Deserializer
VAR_INPUT
	Index : UDINT;
END_VAR
GetElementByIndex := this^;
END_METHOD

METHOD GetKeyArray : I_Deserializer
VAR_INPUT
	Key : T_MAXSTRING;
END_VAR
GetKeyArray := this^;
END_METHOD

METHOD GetKeyObject : I_Deserializer
VAR_INPUT
	Key : T_MAXSTRING;
END_VAR
GetKeyObject := this^;
END_METHOD

METHOD GetObject : I_Deserializer
VAR_INPUT
END_VAR
GetObject := this^;
END_METHOD

METHOD GetObjectEnumerator : I_DeserializerObjectForwardEnumerator
VAR_INPUT
END_VAR
GetObjectEnumerator := CreateNullObjectEnumerator();
END_METHOD

METHOD TryDeserializeKeyToObject : BOOL
VAR_INPUT
	Key : T_MAXSTRING;
	Object : I_Deserializable;
	Feedback : I_DeserializerFeedback;
END_VAR
VAR
	error : I_Error;
END_VAR
IF Key = '' THEN
	error := errorFactory.CreateInvalidKeyError();
	Feedback.LogError(error);
	RETURN;
END_IF

TryDeserializeKeyToObject := FALSE;
END_METHOD

METHOD TryDeserializeToObject : BOOL
VAR_INPUT
	Object : I_Deserializable;
	Feedback : I_DeserializerFeedback;
END_VAR
TryDeserializeToObject := Object.TryDeserializeFrom(THIS^, Feedback);
END_METHOD

METHOD TryGetBase64 : BOOL
VAR_INPUT
	pBytes : POINTER TO BYTE;
	nBytes : DINT;
	Feedback : I_DeserializerFeedback;
END_VAR
VAR
	error : I_Error;
END_VAR
error := errorFactory.CreateIncorrectTypeError('Base64');
Feedback.LogError(error);
END_METHOD

METHOD TryGetBool : BOOL
VAR_INPUT
	Destination : REFERENCE TO BOOL;
	Feedback : I_DeserializerFeedback;
END_VAR
VAR
	error : I_Error;
END_VAR
error := errorFactory.CreateIncorrectTypeError('BOOL');
Feedback.LogError(error);
END_METHOD

METHOD TryGetByte : BOOL
VAR_INPUT
	Destination : REFERENCE TO BYTE;
	Feedback : I_DeserializerFeedback;
END_VAR
VAR
	error : I_Error;
END_VAR
error := errorFactory.CreateIncorrectTypeError('BYTE');
Feedback.LogError(error);
END_METHOD

METHOD TryGetDateTime : BOOL
VAR_INPUT
	Destination : REFERENCE TO DATE_AND_TIME;
	Feedback : I_DeserializerFeedback;
END_VAR
VAR
	error : I_Error;
END_VAR
error := errorFactory.CreateIncorrectTypeError('DATE_AND_TIME');
Feedback.LogError(error);
END_METHOD

METHOD TryGetDcTime : BOOL
VAR_INPUT
	Destination : REFERENCE TO DCTIME;
	Feedback : I_DeserializerFeedback;
END_VAR
VAR
	error : I_Error;
END_VAR
error := errorFactory.CreateIncorrectTypeError('DCTIME');
Feedback.LogError(error);
END_METHOD

METHOD TryGetDint : BOOL
VAR_INPUT
	Destination : REFERENCE TO DINT;
	Feedback : I_DeserializerFeedback;
END_VAR
VAR
	error : I_Error;
END_VAR
error := errorFactory.CreateIncorrectTypeError('DINT');
Feedback.LogError(error);
END_METHOD

METHOD TryGetDword : BOOL
VAR_INPUT
	Destination : REFERENCE TO DWORD;
	Feedback : I_DeserializerFeedback;
END_VAR
VAR
	error : I_Error;
END_VAR
error := errorFactory.CreateIncorrectTypeError('DWORD');
Feedback.LogError(error);
END_METHOD

METHOD TryGetFileTime : BOOL
VAR_INPUT
	Destination : REFERENCE TO FILETIME;
	Feedback : I_DeserializerFeedback;
END_VAR
VAR
	error : I_Error;
END_VAR
error := errorFactory.CreateIncorrectTypeError('FILETIME');
Feedback.LogError(error);
END_METHOD

METHOD TryGetHexAsBytes : BOOL
VAR_INPUT
	pBytes : POINTER TO BYTE;
	nBytes : DINT;
	Feedback : I_DeserializerFeedback;
END_VAR
VAR
	error : I_Error;
END_VAR
error := errorFactory.CreateIncorrectTypeError('HexBinary');
Feedback.LogError(error);
END_METHOD

METHOD TryGetInt : BOOL
VAR_INPUT
	Destination : REFERENCE TO INT;
	Feedback : I_DeserializerFeedback;
END_VAR
VAR
	error : I_Error;
END_VAR
error := errorFactory.CreateIncorrectTypeError('INT');
Feedback.LogError(error);
END_METHOD

METHOD TryGetKeyBase64 : BOOL
VAR_INPUT
	Key : T_MAXSTRING;
	pBytes : POINTER TO BYTE;
	nBytes : DINT;
	Feedback : I_DeserializerFeedback;
END_VAR
VAR
	error : I_Error;
END_VAR
error := errorFactory.CreateIncorrectKeyTypeError('Base64',Key);
Feedback.LogError(error);
END_METHOD

METHOD TryGetKeyBool : BOOL
VAR_INPUT
	Key : T_MAXSTRING;
	Destination : REFERENCE TO BOOL;
	Feedback : I_DeserializerFeedback;
END_VAR
VAR
	error : I_Error;
END_VAR
error := errorFactory.CreateIncorrectKeyTypeError('BOOL',Key);
Feedback.LogError(error);
END_METHOD

METHOD TryGetKeyByte : BOOL
VAR_INPUT
	Key : T_MAXSTRING;
	Destination : REFERENCE TO BYTE;
	Feedback : I_DeserializerFeedback;
END_VAR
VAR
	error : I_Error;
END_VAR
error := errorFactory.CreateIncorrectKeyTypeError('BYTE',Key);
Feedback.LogError(error);
END_METHOD

METHOD TryGetKeyDateTime : BOOL
VAR_INPUT
	Key : T_MAXSTRING;
	Destination : REFERENCE TO DATE_AND_TIME;
	Feedback : I_DeserializerFeedback;
END_VAR
VAR
	error : I_Error;
END_VAR
error := errorFactory.CreateIncorrectKeyTypeError('DATE_AND_TIME',Key);
Feedback.LogError(error);
END_METHOD

METHOD TryGetKeyDcTime : BOOL
VAR_INPUT
	Key : T_MAXSTRING;
	Destination : REFERENCE TO DCTIME;
	Feedback : I_DeserializerFeedback;
END_VAR
VAR
	error : I_Error;
END_VAR
error := errorFactory.CreateIncorrectKeyTypeError('DCTIME',Key);
Feedback.LogError(error);
END_METHOD

METHOD TryGetKeyDint : BOOL
VAR_INPUT
	Key : T_MAXSTRING;
	Destination : REFERENCE TO DINT;
	Feedback : I_DeserializerFeedback;
END_VAR
VAR
	error : I_Error;
END_VAR
error := errorFactory.CreateIncorrectKeyTypeError('DINT',Key);
Feedback.LogError(error);
END_METHOD

METHOD TryGetKeyDword : BOOL
VAR_INPUT
	Key : T_MAXSTRING;
	Destination : REFERENCE TO DWORD;
	Feedback : I_DeserializerFeedback;
END_VAR
VAR
	error : I_Error;
END_VAR
error := errorFactory.CreateIncorrectKeyTypeError('DWORD',Key);
Feedback.LogError(error);
END_METHOD

METHOD TryGetKeyFileTime : BOOL
VAR_INPUT
	Key : T_MAXSTRING;
	Destination : REFERENCE TO FILETIME;
	Feedback : I_DeserializerFeedback;
END_VAR
VAR
	error : I_Error;
END_VAR
error := errorFactory.CreateIncorrectKeyTypeError('FILETIME',Key);
Feedback.LogError(error);
END_METHOD

METHOD TryGetKeyHexAsBytes : BOOL
VAR_INPUT
	Key : T_MAXSTRING;
	pBytes : POINTER TO BYTE;
	nBytes : DINT;
	Feedback : I_DeserializerFeedback;
END_VAR
VAR
	error : I_Error;
END_VAR
error := errorFactory.CreateIncorrectKeyTypeError('HexBinary',Key);
Feedback.LogError(error);
END_METHOD

METHOD TryGetKeyInt : BOOL
VAR_INPUT
	Key : T_MAXSTRING;
	Destination : REFERENCE TO INT;
	Feedback : I_DeserializerFeedback;
END_VAR
VAR
	error : I_Error;
END_VAR
error := errorFactory.CreateIncorrectKeyTypeError('INT',Key);
Feedback.LogError(error);
END_METHOD

METHOD TryGetKeyLint : BOOL
VAR_INPUT
	Key : T_MAXSTRING;
	Destination : REFERENCE TO LINT;
	Feedback : I_DeserializerFeedback;
END_VAR
VAR
	error : I_Error;
END_VAR
error := errorFactory.CreateIncorrectKeyTypeError('LINT',Key);
Feedback.LogError(error);
END_METHOD

METHOD TryGetKeyLreal : BOOL
VAR_INPUT
	Key : T_MAXSTRING;
	Destination : REFERENCE TO LREAL;
	Feedback : I_DeserializerFeedback;
END_VAR
VAR
	error : I_Error;
END_VAR
error := errorFactory.CreateIncorrectKeyTypeError('LREAL',Key);
Feedback.LogError(error);
END_METHOD

METHOD TryGetKeyLtime : BOOL
VAR_INPUT
	Key : T_MAXSTRING;
	Destination : REFERENCE TO LTIME;
	Feedback : I_DeserializerFeedback;
END_VAR
VAR
	error : I_Error;
END_VAR
error := errorFactory.CreateIncorrectKeyTypeError('LTIME',Key);
Feedback.LogError(error);
END_METHOD

METHOD TryGetKeyLword : BOOL
VAR_INPUT
	Key : T_MAXSTRING;
	Destination : REFERENCE TO LWORD;
	Feedback : I_DeserializerFeedback;
END_VAR
VAR
	error : I_Error;
END_VAR
error := errorFactory.CreateIncorrectKeyTypeError('LWORD',Key);
Feedback.LogError(error);
END_METHOD

METHOD TryGetKeyReal : BOOL
VAR_INPUT
	Key : T_MAXSTRING;
	Destination : REFERENCE TO REAL;
	Feedback : I_DeserializerFeedback;
END_VAR
VAR
	error : I_Error;
END_VAR
error := errorFactory.CreateIncorrectKeyTypeError('REAL',Key);
Feedback.LogError(error);
END_METHOD

METHOD TryGetKeySint : BOOL
VAR_INPUT
	Key : T_MAXSTRING;
	Destination : REFERENCE TO SINT;
	Feedback : I_DeserializerFeedback;
END_VAR
VAR
	error : I_Error;
END_VAR
error := errorFactory.CreateIncorrectKeyTypeError('SINT',Key);
Feedback.LogError(error);
END_METHOD

METHOD TryGetKeyString : BOOL
VAR_INPUT
	Key : T_MAXSTRING;
	Destination : REFERENCE TO STRING;
	Feedback : I_DeserializerFeedback;
END_VAR
VAR
	error : I_Error;
END_VAR
error := errorFactory.CreateIncorrectKeyTypeError('STRING',Key);
Feedback.LogError(error);
END_METHOD

METHOD TryGetKeyTime : BOOL
VAR_INPUT
	Key : T_MAXSTRING;
	Destination : REFERENCE TO TIME;
	Feedback : I_DeserializerFeedback;
END_VAR
VAR
	error : I_Error;
END_VAR
error := errorFactory.CreateIncorrectKeyTypeError('TIME',Key);
Feedback.LogError(error);
END_METHOD

METHOD TryGetKeyTod : BOOL
VAR_INPUT
	Key : T_MAXSTRING;
	Destination : REFERENCE TO TOD;
	Feedback : I_DeserializerFeedback;
END_VAR
VAR
	error : I_Error;
END_VAR
error := errorFactory.CreateIncorrectKeyTypeError('TOD',Key);
Feedback.LogError(error);
END_METHOD

METHOD TryGetKeyUdint : BOOL
VAR_INPUT
	Key : T_MAXSTRING;
	Destination : REFERENCE TO UDINT;
	Feedback : I_DeserializerFeedback;
END_VAR
VAR
	error : I_Error;
END_VAR
error := errorFactory.CreateIncorrectKeyTypeError('UDINT',Key);
Feedback.LogError(error);
END_METHOD

METHOD TryGetKeyUint : BOOL
VAR_INPUT
	Key : T_MAXSTRING;
	Destination : REFERENCE TO UINT;
	Feedback : I_DeserializerFeedback;
END_VAR
VAR
	error : I_Error;
END_VAR
error := errorFactory.CreateIncorrectKeyTypeError('UINT',Key);
Feedback.LogError(error);
END_METHOD

METHOD TryGetKeyUlint : BOOL
VAR_INPUT
	Key : T_MAXSTRING;
	Destination : REFERENCE TO ULINT;
	Feedback : I_DeserializerFeedback;
END_VAR
VAR
	error : I_Error;
END_VAR
error := errorFactory.CreateIncorrectKeyTypeError('ULINT',Key);
Feedback.LogError(error);
END_METHOD

METHOD TryGetKeyUsint : BOOL
VAR_INPUT
	Key : T_MAXSTRING;
	Destination : REFERENCE TO USINT;
	Feedback : I_DeserializerFeedback;
END_VAR
VAR
	error : I_Error;
END_VAR
error := errorFactory.CreateIncorrectKeyTypeError('USINT',Key);
Feedback.LogError(error);
END_METHOD

METHOD TryGetKeyWord : BOOL
VAR_INPUT
	Key : T_MAXSTRING;
	Destination : REFERENCE TO WORD;
	Feedback : I_DeserializerFeedback;
END_VAR
VAR
	error : I_Error;
END_VAR
error := errorFactory.CreateIncorrectKeyTypeError('USINT',Key);
Feedback.LogError(error);
END_METHOD

METHOD TryGetLint : BOOL
VAR_INPUT
	Destination : REFERENCE TO LINT;
	Feedback : I_DeserializerFeedback;
END_VAR
VAR
	error : I_Error;
END_VAR
error := errorFactory.CreateIncorrectTypeError('LINT');
Feedback.LogError(error);
END_METHOD

METHOD TryGetLreal : BOOL
VAR_INPUT
	Destination : REFERENCE TO LREAL;
	Feedback : I_DeserializerFeedback;
END_VAR
VAR
	error : I_Error;
END_VAR
error := errorFactory.CreateIncorrectTypeError('LREAL');
Feedback.LogError(error);
END_METHOD

METHOD TryGetLtime : BOOL
VAR_INPUT
	Destination : REFERENCE TO LTIME;
	Feedback : I_DeserializerFeedback;
END_VAR
VAR
	error : I_Error;
END_VAR
error := errorFactory.CreateIncorrectTypeError('LTIME');
Feedback.LogError(error);
END_METHOD

METHOD TryGetLword : BOOL
VAR_INPUT
	Destination : REFERENCE TO LWORD;
	Feedback : I_DeserializerFeedback;
END_VAR
VAR
	error : I_Error;
END_VAR
error := errorFactory.CreateIncorrectTypeError('LWORD');
Feedback.LogError(error);
END_METHOD

METHOD TryGetReal : BOOL
VAR_INPUT
	Destination : REFERENCE TO REAL;
	Feedback : I_DeserializerFeedback;
END_VAR
VAR
	error : I_Error;
END_VAR
error := errorFactory.CreateIncorrectTypeError('REAL');
Feedback.LogError(error);
END_METHOD

METHOD TryGetSint : BOOL
VAR_INPUT
	Destination : REFERENCE TO SINT;
	Feedback : I_DeserializerFeedback;
END_VAR
VAR
	error : I_Error;
END_VAR
error := errorFactory.CreateIncorrectTypeError('SINT');
Feedback.LogError(error);
END_METHOD

METHOD TryGetString : BOOL
VAR_INPUT
	Destination : REFERENCE TO STRING;
	Feedback : I_DeserializerFeedback;
END_VAR
VAR
	error : I_Error;
END_VAR
error := errorFactory.CreateIncorrectTypeError('STRING');
Feedback.LogError(error);
END_METHOD

METHOD TryGetTime : BOOL
VAR_INPUT
	Destination : REFERENCE TO TIME;
	Feedback : I_DeserializerFeedback;
END_VAR
VAR
	error : I_Error;
END_VAR
error := errorFactory.CreateIncorrectTypeError('TIME');
Feedback.LogError(error);
END_METHOD

METHOD TryGetTod : BOOL
VAR_INPUT
	Destination : REFERENCE TO TOD;
	Feedback : I_DeserializerFeedback;
END_VAR
VAR
	error : I_Error;
END_VAR
error := errorFactory.CreateIncorrectTypeError('TOD');
Feedback.LogError(error);
END_METHOD

METHOD TryGetUdint : BOOL
VAR_INPUT
	Destination : REFERENCE TO UDINT;
	Feedback : I_DeserializerFeedback;
END_VAR
VAR
	error : I_Error;
END_VAR
error := errorFactory.CreateIncorrectTypeError('UDINT');
Feedback.LogError(error);
END_METHOD

METHOD TryGetUint : BOOL
VAR_INPUT
	Destination : REFERENCE TO UINT;
	Feedback : I_DeserializerFeedback;
END_VAR
VAR
	error : I_Error;
END_VAR
error := errorFactory.CreateIncorrectTypeError('UINT');
Feedback.LogError(error);
END_METHOD

METHOD TryGetUlint : BOOL
VAR_INPUT
	Destination : REFERENCE TO ULINT;
	Feedback : I_DeserializerFeedback;
END_VAR
VAR
	error : I_Error;
END_VAR
error := errorFactory.CreateIncorrectTypeError('ULINT');
Feedback.LogError(error);
END_METHOD

METHOD TryGetUsint : BOOL
VAR_INPUT
	Destination : REFERENCE TO USINT;
	Feedback : I_DeserializerFeedback;
END_VAR
VAR
	error : I_Error;
END_VAR
error := errorFactory.CreateIncorrectTypeError('USINT');
Feedback.LogError(error);
END_METHOD

METHOD TryGetWord : BOOL
VAR_INPUT
	Destination : REFERENCE TO WORD;
	Feedback : I_DeserializerFeedback;
END_VAR
VAR
	error : I_Error;
END_VAR
error := errorFactory.CreateIncorrectTypeError('WORD');
Feedback.LogError(error);
END_METHOD

END_FUNCTION_BLOCK

// mobject-json/_Internal/JsonDeserializerForwardEnumerator/JsonDeserializerNullArrayForwardEnumerator
{attribute 'linkalways'} 
{attribute 'no_explicit_call' := 'This FB is a CLASS and must be accessed using methods or properties'}
{attribute 'enable_dynamic_creation'}
FUNCTION_BLOCK JsonDeserializerNullArrayForwardEnumerator EXTENDS Disposable IMPLEMENTS I_DeserializerArrayForwardEnumerator, I_EventHandler
VAR
	parent : I_JsonDeserializer;
	nullNode : I_Deserializer;
	invalid : BOOL := FALSE; 
END_VAR

METHOD FB_init : BOOL
VAR_INPUT
	bInitRetains : BOOL; // if TRUE, the retain variables are initialized (warm start / cold start)
	bInCopyCode : BOOL;  // if TRUE, the instance afterwards gets moved into the copy code (online change)
	ParentJsonDeserializer : I_JsonDeserializer;
	ParentNullDeserializer : I_Deserializer;
END_VAR
parent := ParentJsonDeserializer;
nullNode := ParentNullDeserializer;

parent.OnEvent('OnChanged',THIS^);
parent.OnEvent('OnDisposed',THIS^);
END_METHOD

METHOD FB_exit : BOOL
VAR_INPUT
	bInCopyCode : BOOL; // if TRUE, the exit method is called for exiting an instance that is copied afterwards (online change).
END_VAR
IF bInCopyCode THEN
	RETURN;
END_IF

IF parent = 0 THEN
	RETURN;
END_IF

parent.OffEvent('OnChanged',THIS^);
parent.OffEvent('OnDisposed',THIS^);
END_METHOD

PROPERTY PUBLIC Current : I_Deserializer
GET
Current := nullNode;
END_GET
END_PROPERTY

METHOD PUBLIC HandleEvent
VAR_INPUT
	Event : I_Event;
END_VAR
VAR
	changedEvent : I_JsonDeserializerChangedEvent;
	disposedEvent : I_JsonDeserializerDisposedEvent;
END_VAR
IF __QUERYINTERFACE(Event, changedEvent) THEN
	invalid := TRUE;
ELSIF __QUERYINTERFACE(Event, disposedEvent) THEN
	parent := 0;
	Dispose();
END_IF
END_METHOD

PROPERTY Index : DINT
GET
Index := -1;
END_GET
END_PROPERTY

PROPERTY PUBLIC IsValid : BOOL
GET
PUBLIC
IsValid := (NOT invalid AND parent <> 0);
END_GET
END_PROPERTY

METHOD PUBLIC MoveNext : BOOL
MoveNext := FALSE;
END_METHOD

END_FUNCTION_BLOCK

// mobject-json/_Internal/JsonDeserializerForwardEnumerator/JsonDeserializerNullObjectForwardEnumerator
{attribute 'linkalways'} 
{attribute 'no_explicit_call' := 'This FB is a CLASS and must be accessed using methods or properties'}
{attribute 'enable_dynamic_creation'}
FUNCTION_BLOCK JsonDeserializerNullObjectForwardEnumerator EXTENDS Disposable IMPLEMENTS I_DeserializerObjectForwardEnumerator, I_EventHandler
VAR
	parent : I_JsonDeserializer;
	nullNode : I_Deserializer;
	invalid : BOOL := FALSE; 
END_VAR

METHOD FB_init : BOOL
VAR_INPUT
	bInitRetains : BOOL; // if TRUE, the retain variables are initialized (warm start / cold start)
	bInCopyCode : BOOL;  // if TRUE, the instance afterwards gets moved into the copy code (online change)
	ParentJsonDeserializer : I_JsonDeserializer;
	ParentNullDeserializer : I_Deserializer;
END_VAR
parent := ParentJsonDeserializer;
nullNode := ParentNullDeserializer;

parent.OnEvent('OnChanged',THIS^);
parent.OnEvent('OnDisposed',THIS^);
END_METHOD

METHOD FB_exit : BOOL
VAR_INPUT
	bInCopyCode : BOOL; // if TRUE, the exit method is called for exiting an instance that is copied afterwards (online change).
END_VAR
IF bInCopyCode THEN
	RETURN;
END_IF

IF parent = 0 THEN
	RETURN;
END_IF

parent.OffEvent('OnChanged',THIS^);
parent.OffEvent('OnDisposed',THIS^);
END_METHOD

PROPERTY PUBLIC Current : I_Deserializer
GET
Current := nullNode;
END_GET
END_PROPERTY

METHOD PUBLIC HandleEvent
VAR_INPUT
	Event : I_Event;
END_VAR
VAR
	changedEvent : I_JsonDeserializerChangedEvent;
	disposedEvent : I_JsonDeserializerDisposedEvent;
END_VAR
IF __QUERYINTERFACE(Event, changedEvent) THEN
	invalid := TRUE;
ELSIF __QUERYINTERFACE(Event, disposedEvent) THEN
	parent := 0;
	Dispose();
END_IF
END_METHOD

PROPERTY PUBLIC IsValid : BOOL
GET
PUBLIC
IsValid := (NOT invalid AND parent <> 0);
END_GET
END_PROPERTY

PROPERTY Key : T_MAXSTRING
GET
END_GET
END_PROPERTY

METHOD PUBLIC MoveNext : BOOL
MoveNext := FALSE;
END_METHOD

END_FUNCTION_BLOCK

// mobject-json/JsonSerializer/JsonSerializer
{attribute 'linkalways'} 
{attribute 'no_explicit_call' := 'This FB is a CLASS and must be accessed using methods or properties'}
{attribute 'enable_dynamic_creation'}
FUNCTION_BLOCK JsonSerializer EXTENDS Disposable IMPLEMENTS I_Serializer;
VAR
	jsonSaxWriter : FB_JsonSaxWriter;
END_VAR

METHOD FB_exit : BOOL
VAR_INPUT
	bInCopyCode : BOOL; // if TRUE, the exit method is called for exiting an instance that is copied afterwards (online change).
END_VAR
IF bInCopyCode THEN
	RETURN;
END_IF

jsonSaxWriter.ResetDocument();
END_METHOD

METHOD PUBLIC AddBase64 : I_Serializer
VAR_INPUT
	pBytes : POINTER TO BYTE;
	nBytes : DINT;
END_VAR
jsonSaxWriter.AddBase64(pBytes, nBytes);
AddBase64 := THIS^;
END_METHOD

METHOD PUBLIC AddBool : I_Serializer
VAR_INPUT
	Value : BOOL;
END_VAR
jsonSaxWriter.AddBool(Value);
AddBool := THIS^;
END_METHOD

METHOD PUBLIC AddByte : I_Serializer
VAR_INPUT
	Value : BYTE;
END_VAR
jsonSaxWriter.AddUDint(BYTE_TO_UDINT(Value));
AddByte := THIS^;
END_METHOD

METHOD PUBLIC AddBytesAsHex : I_Serializer
VAR_INPUT
	pBytes : POINTER TO BYTE;
	nBytes : DINT;
END_VAR
jsonSaxWriter.AddHexBinary(pBytes, nBytes);
AddBytesAsHex := THIS^;
END_METHOD

METHOD PUBLIC AddDateTime : I_Serializer
VAR_INPUT
	Value : DATE_AND_TIME;
END_VAR
jsonSaxWriter.AddDateTime(Value);
AddDateTime := THIS^;
END_METHOD

METHOD PUBLIC AddDcTime : I_Serializer
VAR_INPUT
	Value : DCTIME;
END_VAR
jsonSaxWriter.AddDcTime(Value);
AddDcTime := THIS^;
END_METHOD

METHOD PUBLIC AddDint : I_Serializer
VAR_INPUT
	Value : DINT;
END_VAR
jsonSaxWriter.AddDint(Value);
AddDint := THIS^;
END_METHOD

METHOD PUBLIC AddDword : I_Serializer
VAR_INPUT
	Value : DWORD;
END_VAR
jsonSaxWriter.AddUDint(DWORD_TO_UDINT(Value));
AddDword := THIS^;
END_METHOD

METHOD PUBLIC AddFileTime : I_Serializer
VAR_INPUT
	Value : FILETIME;
END_VAR
jsonSaxWriter.AddFileTime(Value);
AddFileTime := THIS^;
END_METHOD

METHOD PUBLIC AddInt : I_Serializer
VAR_INPUT
	Value : INT;
END_VAR
jsonSaxWriter.AddDint(INT_TO_DINT(Value));
AddInt := THIS^;
END_METHOD

METHOD PUBLIC AddKey : I_Serializer
VAR_INPUT
	Key : T_MAXSTRING;
END_VAR
jsonSaxWriter.AddKey(Key);
AddKey := THIS^;
END_METHOD

METHOD PUBLIC AddKeyBase64 : I_Serializer
VAR_INPUT
	Key : T_MAXSTRING;
	pBytes : POINTER TO BYTE;
	nBytes : DINT;
END_VAR
AddKey(Key);
AddBase64(pBytes, nBytes);
AddKeyBase64 := THIS^;
END_METHOD

METHOD PUBLIC AddKeyBool : I_Serializer
VAR_INPUT
	Key : T_MAXSTRING;
	Value : BOOL;
END_VAR
AddKey(Key);
AddBool(Value);
AddKeyBool := THIS^;
END_METHOD

METHOD PUBLIC AddKeyByte : I_Serializer
VAR_INPUT
	Key : T_MAXSTRING;
	Value : BYTE;
END_VAR
AddKey(Key);
AddByte(Value);
AddKeyByte := THIS^;
END_METHOD

METHOD PUBLIC AddKeyBytesAsHex : I_Serializer
VAR_INPUT
	Key : T_MAXSTRING;
	pBytes : POINTER TO BYTE;
	nBytes : DINT;
END_VAR
AddKey(Key);
AddBytesAsHex(pBytes, nBytes);
AddKeyBytesAsHex := THIS^;
END_METHOD

METHOD PUBLIC AddKeyDateTime : I_Serializer
VAR_INPUT
	Key : T_MAXSTRING;
	Value : DATE_AND_TIME;
END_VAR
AddKey(Key);
AddDateTime(Value);
AddKeyDateTime := THIS^;
END_METHOD

METHOD PUBLIC AddKeyDcTime : I_Serializer
VAR_INPUT
	Key : T_MAXSTRING;
	Value : DCTIME;
END_VAR
AddKey(Key);
AddDcTime(Value);
AddKeyDcTime := THIS^;
END_METHOD

METHOD PUBLIC AddKeyDint : I_Serializer
VAR_INPUT
	Key : T_MAXSTRING;
	Value : DINT;
END_VAR
AddKey(Key);
AddDint(Value);
AddKeyDint := THIS^;
END_METHOD

METHOD PUBLIC AddKeyDword : I_Serializer
VAR_INPUT
	Key : T_MAXSTRING;
	Value : DWORD;
END_VAR
AddKey(Key);
AddDword(Value);
AddKeyDword := THIS^;
END_METHOD

METHOD PUBLIC AddKeyFileTime : I_Serializer
VAR_INPUT
	Key : T_MAXSTRING;
	Value : FILETIME;
END_VAR
AddKey(Key);
AddFileTime(Value);
AddKeyFileTime := THIS^;
END_METHOD

METHOD PUBLIC AddKeyInt : I_Serializer
VAR_INPUT
	Key : T_MAXSTRING;
	Value : INT;
END_VAR
AddKey(Key);
AddInt(Value);
AddKeyInt := THIS^;
END_METHOD

METHOD PUBLIC AddKeyLint : I_Serializer
VAR_INPUT
	Key : T_MAXSTRING;
	Value : LINT;
END_VAR
AddKey(Key);
AddLint(Value);
AddKeyLint := THIS^;
END_METHOD

METHOD PUBLIC AddKeyLreal : I_Serializer
VAR_INPUT
	Key : T_MAXSTRING;
	Value : LREAL;
END_VAR
AddKey(Key);
AddLreal(Value);
AddKeyLreal := THIS^;
END_METHOD

METHOD PUBLIC AddKeyLtime : I_Serializer
VAR_INPUT
	Key : T_MAXSTRING;
	Value : LTIME;
END_VAR
AddKey(Key);
AddLTIME(Value);
AddKeyLtime := THIS^;
END_METHOD

METHOD PUBLIC AddKeyLword : I_Serializer
VAR_INPUT
	Key : T_MAXSTRING;
	Value : LWORD;
END_VAR
AddKey(Key);
AddLword(Value);
AddKeyLword := THIS^;
END_METHOD

METHOD PUBLIC AddKeyNull : I_Serializer
VAR_INPUT
	Key : T_MAXSTRING;
END_VAR
AddKey(Key);
AddNull();
AddKeyNull := THIS^;
END_METHOD

METHOD PUBLIC AddKeyObject : I_Serializer
VAR_INPUT
	Key : T_MAXSTRING;
	Object : I_Serializable;
END_VAR
AddKey(Key);
Object.SerializeWith(THIS^);
AddKeyObject := THIS^;
END_METHOD

METHOD PUBLIC AddKeyRawJson : I_Serializer
VAR_INPUT
	Key : T_MAXSTRING;
	RawObject : REFERENCE TO STRING;;
END_VAR
AddKey(Key);
AddRawJson(RawObject);
AddKeyRawJson := THIS^;
END_METHOD

METHOD PUBLIC AddKeyReal : I_Serializer
VAR_INPUT
	Key : T_MAXSTRING;
	Value : REAL;
END_VAR
AddKey(Key);
AddReal(Value);
AddKeyReal := THIS^;
END_METHOD

METHOD PUBLIC AddKeySint : I_Serializer
VAR_INPUT
	Key : T_MAXSTRING;
	Value : SINT;
END_VAR
AddKey(Key);
AddSint(Value);
AddKeySint := THIS^;
END_METHOD

METHOD PUBLIC AddKeyString : I_Serializer
VAR_INPUT
	Key : T_MAXSTRING;
	Value : T_MAXSTRING;
END_VAR
AddKey(Key);
AddString(Value);
AddKeyString := THIS^;
END_METHOD

METHOD PUBLIC AddKeyStringByRef : I_Serializer
VAR_INPUT
	Key : T_MAXSTRING;
	Value : REFERENCE TO STRING;;
END_VAR
AddKey(Key);
AddStringByRef(Value);
AddKeyStringByRef := THIS^;
END_METHOD

METHOD PUBLIC AddKeyTime : I_Serializer
VAR_INPUT
	Key : T_MAXSTRING;
	Value : TIME;
END_VAR
AddKey(Key);
AddTime(Value);
AddKeyTime := THIS^;
END_METHOD

METHOD PUBLIC AddKeyTod : I_Serializer
VAR_INPUT
	Key : T_MAXSTRING;
	Value : TOD;
END_VAR
AddKey(Key);
AddTod(Value);
AddKeyTod := THIS^;
END_METHOD

METHOD PUBLIC AddKeyUdint : I_Serializer
VAR_INPUT
	Key : T_MAXSTRING;
	Value : UDINT;
END_VAR
AddKey(Key);
AddUdint(Value);
AddKeyUdint := THIS^;
END_METHOD

METHOD PUBLIC AddKeyUint : I_Serializer
VAR_INPUT
	Key : T_MAXSTRING;
	Value : UINT;
END_VAR
AddKey(Key);
AddUint(Value);
AddKeyUint := THIS^;
END_METHOD

METHOD PUBLIC AddKeyUlint : I_Serializer
VAR_INPUT
	Key : T_MAXSTRING;
	Value : ULINT;
END_VAR
AddKey(Key);
AddUlint(Value);
AddKeyUlint := THIS^;
END_METHOD

METHOD PUBLIC AddKeyUsint : I_Serializer
VAR_INPUT
	Key : T_MAXSTRING;
	Value : USINT;
END_VAR
AddKey(Key);
AddUsint(Value);
AddKeyUsint := THIS^;
END_METHOD

METHOD PUBLIC AddKeyWord : I_Serializer
VAR_INPUT
	Key : T_MAXSTRING;
	Value : WORD;
END_VAR
AddKey(Key);
AddWord(Value);
AddKeyWord := THIS^;
END_METHOD

METHOD PUBLIC AddLint : I_Serializer
VAR_INPUT
	Value : LINT;
END_VAR
jsonSaxWriter.AddLint(Value);
AddLint := THIS^;
END_METHOD

METHOD PUBLIC AddLreal : I_Serializer
VAR_INPUT
	Value : LREAL;
END_VAR
jsonSaxWriter.AddLreal(Value);
AddLreal := THIS^;
END_METHOD

METHOD PUBLIC AddLtime : I_Serializer
VAR_INPUT
	Value : LTIME;
END_VAR
VAR
	converted : T_MAXSTRING;
END_VAR
converted := LTIME_TO_STRING(Value);
jsonSaxWriter.AddString(converted);
AddLtime := THIS^;
END_METHOD

METHOD PUBLIC AddLword : I_Serializer
VAR_INPUT
	Value : LWORD;
END_VAR
jsonSaxWriter.AddUlint(LWORD_TO_ULINT(Value));
AddLword := THIS^;
END_METHOD

METHOD PUBLIC AddNull : I_Serializer
VAR_INPUT
END_VAR
jsonSaxWriter.AddNull();
AddNull := THIS^;
END_METHOD

METHOD PUBLIC AddObject
VAR_INPUT
	Object : I_Serializable;
END_VAR
Object.SerializeWith(This^);
END_METHOD

METHOD PUBLIC AddRawJson
VAR_INPUT
	RawObject : REFERENCE TO STRING;
END_VAR
jsonSaxWriter.AddRawObject(RawObject);
END_METHOD

METHOD PUBLIC AddReal : I_Serializer
VAR_INPUT
	Value : REAL;
END_VAR
// real to lreal is used to negate an issue with TC4024.55 which prevents max REAL from being serailized.  
// so a REAL_TO_LREAL conversion is made to ensure this is always possible.  
jsonSaxWriter.AddLReal(REAL_TO_LREAL(Value));
AddReal := THIS^;
END_METHOD

METHOD PUBLIC AddSint : I_Serializer
VAR_INPUT
	Value : SINT;
END_VAR
jsonSaxWriter.AddDint(SINT_TO_DINT(Value));
AddSint := THIS^;
END_METHOD

METHOD PUBLIC AddString : I_Serializer
VAR_INPUT
	Value : T_MAXSTRING;
END_VAR
jsonSaxWriter.AddString(Value);
AddString := THIS^;
END_METHOD

METHOD PUBLIC AddStringByRef : I_Serializer
VAR_INPUT
	Value : REFERENCE TO STRING;
END_VAR
jsonSaxWriter.AddString(Value);
AddStringByRef := THIS^;
END_METHOD

METHOD PUBLIC AddTime : I_Serializer
VAR_INPUT
	Value : TIME;
END_VAR
VAR
	converted : T_MAXSTRING;
END_VAR
converted := TIME_TO_STRING(Value);
jsonSaxWriter.AddString(converted);
AddTime := THIS^;
END_METHOD

METHOD PUBLIC AddTod : I_Serializer
VAR_INPUT
	Value : TOD;
END_VAR
VAR
	converted : T_MAXSTRING;
END_VAR
converted := TOD_TO_STRING(Value);
jsonSaxWriter.AddString(converted);
AddTod := THIS^;
END_METHOD

METHOD PUBLIC AddUdint : I_Serializer
VAR_INPUT
	Value : UDINT;
END_VAR
jsonSaxWriter.AddUdint(Value);
AddUdint := THIS^;
END_METHOD

METHOD PUBLIC AddUint : I_Serializer
VAR_INPUT
	Value : UINT;
END_VAR
jsonSaxWriter.AddDint(UINT_TO_DINT(Value));
AddUint := THIS^;
END_METHOD

METHOD PUBLIC AddUlint : I_Serializer
VAR_INPUT
	Value : ULINT;
END_VAR
jsonSaxWriter.AddUlint(Value);
AddUlint := THIS^;
END_METHOD

METHOD PUBLIC AddUsint : I_Serializer
VAR_INPUT
	Value : USINT;
END_VAR
jsonSaxWriter.AddDint(USINT_TO_DINT(Value));
AddUsint := THIS^;
END_METHOD

METHOD PUBLIC AddWord : I_Serializer
VAR_INPUT
	Value : WORD;
END_VAR
jsonSaxWriter.AddUDint(WORD_TO_UDINT(Value));
AddWord := THIS^;
END_METHOD

METHOD PUBLIC Clone : I_Serializer
VAR
	pClone : POINTER TO JsonSerializer;
	jsonSize : UDINT;
	pJsonString : POINTER TO STRING;
END_VAR
pClone := __NEW(JsonSerializer);
Clone := pClone^;

jsonSize := jsonSaxWriter.GetDocumentLength();

IF jsonSize = 0 THEN
	// no further cloning to do. 
	RETURN;
END_IF

pJsonString := __NEW(BYTE, jsonSize);

IF jsonSaxWriter.CopyDocument(pJsonString^, jsonSize) = 0 THEN
	__DELETE(pJsonString);
	RETURN;
END_IF

pClone^.AddRawJson(pJsonString^);
__DELETE(pJsonString);
END_METHOD

METHOD PUBLIC EndArray : I_Serializer
VAR_INPUT
END_VAR
jsonSaxWriter.EndArray();
EndArray := THIS^;
END_METHOD

METHOD PUBLIC EndObject : I_Serializer
VAR_INPUT
END_VAR
jsonSaxWriter.EndObject();
EndObject := THIS^;
END_METHOD

METHOD PUBLIC GetSerializedDataLength : UDINT
VAR_INPUT
END_VAR
GetSerializedDataLength := jsonSaxWriter.GetDocumentLength();
END_METHOD

METHOD PUBLIC Reset
VAR_INPUT
END_VAR
jsonSaxWriter.ResetDocument();
END_METHOD

METHOD PUBLIC StartArray : I_Serializer
VAR_INPUT
END_VAR
jsonSaxWriter.StartArray();
StartArray := THIS^;
END_METHOD

METHOD PUBLIC StartObject : I_Serializer
VAR_INPUT
END_VAR
jsonSaxWriter.StartObject();
StartObject := THIS^;
END_METHOD

METHOD TryCopySerializedData : BOOL
VAR_INPUT
	DestinationAddress : PVOID;
	DestinationSize : UDINT;
END_VAR
VAR
	pString : POINTER TO STRING;
END_VAR
pString := DestinationAddress;
TryCopySerializedData := jsonSaxWriter.CopyDocument(pString^, DestinationSize) > 0;
END_METHOD

METHOD TryGetSerializedData : BOOL
VAR_INPUT
	DestinationAddress : PVOID;
	DestinationSize : UDINT;
END_VAR
VAR
	pString : POINTER TO STRING;
END_VAR
pString := DestinationAddress;

IF jsonSaxWriter.CopyDocument(pString^, DestinationSize) = 0 THEN
	RETURN;
END_IF

jsonSaxWriter.ResetDocument();
TryGetSerializedData := TRUE;
END_METHOD

END_FUNCTION_BLOCK
